LIN {X 0,Y 100.276,Z 426.301,A -85,B 0,C 180,E1 -26714.761,E2 -26714.761} C_VEL
LIN {X 0,Y 99.37,Z 433.159,A -85,B 0,C 180,E1 -26720.842,E2 -26720.842} C_VEL
LIN {X 0,Y 99.45,Z 437.817,A -85,B 0,C 180,E1 -26725.946,E2 -26725.946} C_VEL
LIN {X 0,Y 99.702,Z 440.8,A -85,B 0,C 180,E1 -26729.999,E2 -26729.999} C_VEL
LIN {X 0,Y 99.27,Z 443.094,A -85,B 0,C 180,E1 -26734.059,E2 -26734.059} C_VEL
LIN {X 0,Y 99.023,Z 444.925,A -85,B 0,C 180,E1 -26738.159,E2 -26738.159} C_VEL
LIN {X 0,Y 99.917,Z 447.345,A -85,B 0,C 180,E1 -26746.34,E2 -26746.34} C_VEL
LIN {X 0,Y 102.956,Z 448.359,A -85,B 0,C 180,E1 -26754.177,E2 -26754.177} C_VEL
LIN {X 0,Y 108.06,Z 448.023,A -85,B 0,C 180,E1 -26761.351,E2 -26761.351} C_VEL
LIN {X 0,Y 111.325,Z 447.297,A -85,B 0,C 180,E1 -26764.844,E2 -26764.844} C_VEL
LIN {X 0,Y 118.698,Z 444.902,A -85,B 0,C 180,E1 -26770.639,E2 -26770.639} C_VEL
LIN {X 0,Y 127.654,Z 441.015,A -85,B 0,C 180,E1 -26775.701,E2 -26775.701} C_VEL
LIN {X 0,Y 135.078,Z 437.071,A -85,B 0,C 180,E1 -26778.974,E2 -26778.974} C_VEL
LIN {X 0,Y 142.954,Z 432.141,A -85,B 0,C 180,E1 -26781.868,E2 -26781.868} C_VEL
LIN {X 0,Y 152.719,Z 424.964,A -85,B 0,C 180,E1 -26784.769,E2 -26784.769} C_VEL
LIN {X 0,Y 161.484,Z 417.418,A -85,B 0,C 180,E1 -26786.906,E2 -26786.906} C_VEL
LIN {X 0,Y 170.55,Z 408.157,A -85,B 0,C 180,E1 -26788.766,E2 -26788.766} C_VEL
LIN {X 0,Y 179.159,Z 397.683,A -85,B 0,C 180,E1 -26790.216,E2 -26790.216} C_VEL
LIN {X 0,Y 187.164,Z 385.927,A -85,B 0,C 180,E1 -26791.369,E2 -26791.369} C_VEL
LIN {X 0,Y 193.611,Z 374.263,A -85,B 0,C 180,E1 -26792.226,E2 -26792.226} C_VEL
LIN {X 0,Y 199.333,Z 361.205,A -85,B 0,C 180,E1 -26792.895,E2 -26792.895} C_VEL
LIN {X 0,Y 200.129,Z 359.001,A -85,B 0,C 180,E1 -26792.986,E2 -26792.986} C_VEL
LIN {X 0,Y 200.135,Z 358.847,A -85,B 0,C 180,E1 -26793.242,E2 -26793.242} C_VEL
LIN {X 0,Y 199.484,Z 360.339,A -85,B 0,C 180,E1 -26793.791,E2 -26793.791} C_VEL
LIN {X 0,Y 198.376,Z 362.917,A -85,B 0,C 180,E1 -26794.295,E2 -26794.295} C_VEL
LIN {X 0,Y 195.362,Z 369.602,A -85,B 0,C 180,E1 -26795.081,E2 -26795.081} C_VEL
LIN {X 0,Y 191.94,Z 376.275,A -85,B 0,C 180,E1 -26795.732,E2 -26795.732} C_VEL
LIN {X 0,Y 185.418,Z 386.983,A -85,B 0,C 180,E1 -26796.812,E2 -26796.812} C_VEL
LIN {X 0,Y 177.571,Z 397.49,A -85,B 0,C 180,E1 -26798.219,E2 -26798.219} C_VEL
LIN {X 0,Y 168.913,Z 406.976,A -85,B 0,C 180,E1 -26799.961,E2 -26799.961} C_VEL
LIN {X 0,Y 159.727,Z 415.31,A -85,B 0,C 180,E1 -26802.061,E2 -26802.061} C_VEL
LIN {X 0,Y 150.644,Z 422.152,A -85,B 0,C 180,E1 -26804.439,E2 -26804.439} C_VEL
LIN {X 0,Y 141.958,Z 427.534,A -85,B 0,C 180,E1 -26807.126,E2 -26807.126} C_VEL
LIN {X 0,Y 132.044,Z 432.427,A -85,B 0,C 180,E1 -26810.812,E2 -26810.812} C_VEL
LIN {X 0,Y 125.872,Z 434.856,A -85,B 0,C 180,E1 -26813.588,E2 -26813.588} C_VEL
LIN {X 0,Y 119.656,Z 436.729,A -85,B 0,C 180,E1 -26816.841,E2 -26816.841} C_VEL
LIN {X 0,Y 112.482,Z 438.152,A -85,B 0,C 180,E1 -26821.437,E2 -26821.437} C_VEL
LIN {X 0,Y 105.078,Z 438.534,A -85,B 0,C 180,E1 -26827.687,E2 -26827.687} C_VEL
LIN {X 0,Y 100.769,Z 437.945,A -85,B 0,C 180,E1 -26832.475,E2 -26832.475} C_VEL
LIN {X 0,Y 96.542,Z 436.3,A -85,B 0,C 180,E1 -26838.854,E2 -26838.854} C_VEL
LIN {X 0,Y 93.138,Z 433.039,A -85,B 0,C 180,E1 -26846.92,E2 -26846.92} C_VEL
LIN {X 0,Y 91.475,Z 428.303,A -85,B 0,C 180,E1 -26855.182,E2 -26855.182} C_VEL
LIN {X 0,Y 91.387,Z 423.638,A -85,B 0,C 180,E1 -26861.508,E2 -26861.508} C_VEL
LIN {X 0,Y 92.227,Z 417.856,A -85,B 0,C 180,E1 -26867.807,E2 -26867.807} C_VEL
LIN {X 0,Y 93.74,Z 410.783,A -85,B 0,C 180,E1 -26873.954,E2 -26873.954} C_VEL
LIN {X 0,Y 96.114,Z 401.66,A -85,B 0,C 180,E1 -26880.167,E2 -26880.167} C_VEL
LIN {X 0,Y 98.865,Z 392.134,A -85,B 0,C 180,E1 -26885.194,E2 -26885.194} C_VEL
LIN {X 0,Y 102.107,Z 380.518,A -85,B 0,C 180,E1 -26889.871,E2 -26889.871} C_VEL
LIN {X 0,Y 105.174,Z 368.48,A -85,B 0,C 180,E1 -26893.543,E2 -26893.543} C_VEL
LIN {X 0,Y 107.957,Z 355.625,A -85,B 0,C 180,E1 -26896.428,E2 -26896.428} C_VEL
LIN {X 0,Y 110.286,Z 342.25,A -85,B 0,C 180,E1 -26898.577,E2 -26898.577} C_VEL
LIN {X 0,Y 111.831,Z 328.48,A -85,B 0,C 180,E1 -26900.056,E2 -26900.056} C_VEL
LIN {X 0,Y 115.307,Z 288.804,A -85,B 0,C 180,E1 -26902.945,E2 -26902.945} C_VEL
LIN {X 0,Y 108.992,Z 272.53,A -85,B 0,C 180,E1 -26906.42,E2 -26906.42} C_VEL
LIN {X 0,Y 104.471,Z 262.113,A -85,B 0,C 180,E1 -26909.085,E2 -26909.085} C_VEL
LIN {X 0,Y 98.736,Z 250.528,A -85,B 0,C 180,E1 -26912.663,E2 -26912.663} C_VEL
LIN {X 0,Y 96.221,Z 246.747,A -85,B 0,C 180,E1 -26914.262,E2 -26914.262} C_VEL
LIN {X 0,Y 94.549,Z 244.182,A -85,B 0,C 180,E1 -26915.399,E2 -26915.399} C_VEL
LIN {X 0,Y 94.223,Z 242.747,A -85,B 0,C 180,E1 -26915.888,E2 -26915.888} C_VEL
LIN {X 0,Y 94.067,Z 242.767,A -85,B 0,C 180,E1 -26922.953,E2 -26922.953} C_VEL
LIN {X 0,Y 93.79,Z 242.798,A -85,B 0,C 180,E1 -26927.443,E2 -26927.443} C_VEL
LIN {X 0,Y 93.693,Z 242.786,A -85,B 0,C 180,E1 -26932.029,E2 -26932.029} C_VEL
LIN {X 0,Y 93.62,Z 242.82,A -85,B 0,C 180,E1 -26936.772,E2 -26936.772} C_VEL
LIN {X 0,Y 93.584,Z 242.8,A -85,B 0,C 180,E1 -26944.302,E2 -26944.302} C_VEL
LIN {X 0,Y 93.528,Z 242.815,A -85,B 0,C 180,E1 -26952.556,E2 -26952.556} C_VEL
LIN {X 0,Y 93.532,Z 242.834,A -85,B 0,C 180,E1 -26958.714,E2 -26958.714} C_VEL
LIN {X 0,Y 93.585,Z 242.821,A -85,B 0,C 180,E1 -26965.699,E2 -26965.699} C_VEL
LIN {X 0,Y 93.67,Z 242.801,A -85,B 0,C 180,E1 -26974.207,E2 -26974.207} C_VEL
LIN {X 0,Y 93.694,Z 242.81,A -85,B 0,C 180,E1 -26977.973,E2 -26977.973} C_VEL
LIN {X 0,Y 94.045,Z 242.733,A -85,B 0,C 180,E1 -26987.045,E2 -26987.045} C_VEL
LIN {X 0,Y 94.138,Z 242.707,A -85,B 0,C 180,E1 -26991.413,E2 -26991.413} C_VEL
LIN {X 0,Y 94.759,Z 242.681,A -85,B 0,C 180,E1 -27000,E2 -27000} C_VEL
LIN {X 0,Y 94.136,Z 242.725,A -85,B 0,C 180,E1 -27008.588,E2 -27008.588} C_VEL
LIN {X 0,Y 93.962,Z 242.78,A -85,B 0,C 180,E1 -27013.498,E2 -27013.498} C_VEL
LIN {X 0,Y 93.655,Z 242.802,A -85,B 0,C 180,E1 -27022.038,E2 -27022.038} C_VEL
LIN {X 0,Y 93.6,Z 242.83,A -85,B 0,C 180,E1 -27026.777,E2 -27026.777} C_VEL
LIN {X 0,Y 93.581,Z 242.953,A -85,B 0,C 180,E1 -27030.46,E2 -27030.46} C_VEL
LIN {X 0,Y 94.612,Z 245.714,A -85,B 0,C 180,E1 -27031.331,E2 -27031.331} C_VEL
LIN {X 0,Y 96.125,Z 247.852,A -85,B 0,C 180,E1 -27032.322,E2 -27032.322} C_VEL
LIN {X 0,Y 102.127,Z 258.497,A -85,B 0,C 180,E1 -27036.133,E2 -27036.133} C_VEL
LIN {X 0,Y 107.329,Z 272.747,A -85,B 0,C 180,E1 -27039.577,E2 -27039.577} C_VEL
LIN {X 0,Y 112.457,Z 289.346,A -85,B 0,C 180,E1 -27042.816,E2 -27042.816} C_VEL
LIN {X 0,Y 113.674,Z 316.74,A -85,B 0,C 180,E1 -27045.754,E2 -27045.754} C_VEL
LIN {X 0,Y 110.773,Z 348.84,A -85,B 0,C 180,E1 -27048.226,E2 -27048.226} C_VEL
LIN {X 0,Y 108.763,Z 363.104,A -85,B 0,C 180,E1 -27050.047,E2 -27050.047} C_VEL
LIN {X 0,Y 106.272,Z 375.199,A -85,B 0,C 180,E1 -27052.284,E2 -27052.284} C_VEL
LIN {X 0,Y 103.156,Z 387.718,A -85,B 0,C 180,E1 -27055.473,E2 -27055.473} C_VEL
LIN {X 0,Y 99.991,Z 399.014,A -85,B 0,C 180,E1 -27059.363,E2 -27059.363} C_VEL
LIN {X 0,Y 96.926,Z 409.601,A -85,B 0,C 180,E1 -27064.21,E2 -27064.21} C_VEL
LIN {X 0,Y 94.678,Z 418.278,A -85,B 0,C 180,E1 -27069.353,E2 -27069.353} C_VEL
LIN {X 0,Y 92.992,Z 426.684,A -85,B 0,C 180,E1 -27075.78,E2 -27075.78} C_VEL
LIN {X 0,Y 92.35,Z 434.065,A -85,B 0,C 180,E1 -27083.104,E2 -27083.104} C_VEL
LIN {X 0,Y 92.698,Z 439.38,A -85,B 0,C 180,E1 -27089.999,E2 -27089.999} C_VEL
LIN {X 0,Y 92.287,Z 441.774,A -85,B 0,C 180,E1 -27094.366,E2 -27094.366} C_VEL
LIN {X 0,Y 92.291,Z 445.203,A -85,B 0,C 180,E1 -27103.205,E2 -27103.205} C_VEL
LIN {X 0,Y 94.534,Z 447.195,A -85,B 0,C 180,E1 -27111.82,E2 -27111.82} C_VEL
LIN {X 0,Y 99.083,Z 447.77,A -85,B 0,C 180,E1 -27119.768,E2 -27119.768} C_VEL
LIN {X 0,Y 105.387,Z 446.981,A -85,B 0,C 180,E1 -27126.882,E2 -27126.882} C_VEL
LIN {X 0,Y 113.406,Z 444.856,A -85,B 0,C 180,E1 -27132.975,E2 -27132.975} C_VEL
LIN {X 0,Y 122.808,Z 441.311,A -85,B 0,C 180,E1 -27138.069,E2 -27138.069} C_VEL
LIN {X 0,Y 133.255,Z 436.16,A -85,B 0,C 180,E1 -27142.289,E2 -27142.289} C_VEL
LIN {X 0,Y 141.558,Z 431.209,A -85,B 0,C 180,E1 -27145.002,E2 -27145.002} C_VEL
LIN {X 0,Y 151.742,Z 424.029,A -85,B 0,C 180,E1 -27147.698,E2 -27147.698} C_VEL
LIN {X 0,Y 160.865,Z 416.375,A -85,B 0,C 180,E1 -27149.637,E2 -27149.637} C_VEL
LIN {X 0,Y 170.215,Z 407.055,A -85,B 0,C 180,E1 -27151.328,E2 -27151.328} C_VEL
LIN {X 0,Y 179.048,Z 396.59,A -85,B 0,C 180,E1 -27152.632,E2 -27152.632} C_VEL
LIN {X 0,Y 186.418,Z 386.056,A -85,B 0,C 180,E1 -27153.556,E2 -27153.556} C_VEL
LIN {X 0,Y 192.996,Z 374.507,A -85,B 0,C 180,E1 -27154.326,E2 -27154.326} C_VEL
LIN {X 0,Y 196.724,Z 366.706,A -85,B 0,C 180,E1 -27154.693,E2 -27154.693} C_VEL
LIN {X 0,Y 196.816,Z 366.436,A -85,B 0,C 180,E1 -27154.942,E2 -27154.942} C_VEL
LIN {X 0,Y 191.94,Z 376.275,A -85,B 0,C 180,E1 -27155.732,E2 -27155.732} C_VEL
LIN {X 0,Y 188.861,Z 381.616,A -85,B 0,C 180,E1 -27156.025,E2 -27156.025} C_VEL
LIN {X 0,Y 183.135,Z 390.296,A -85,B 0,C 180,E1 -27156.019,E2 -27156.019} C_VEL
LIN {X 0,Y 176.926,Z 398.26,A -85,B 0,C 180,E1 -27156.115,E2 -27156.115} C_VEL
LIN {X 0,Y 173.08,Z 402.614,A -85,B 0,C 180,E1 -27156.583,E2 -27156.583} C_VEL
LIN {X 0,Y 164.976,Z 410.619,A -85,B 0,C 180,E1 -27158.114,E2 -27158.114} C_VEL
LIN {X 0,Y 156.76,Z 417.411,A -85,B 0,C 180,E1 -27159.85,E2 -27159.85} C_VEL
LIN {X 0,Y 146.429,Z 424.498,A -85,B 0,C 180,E1 -27162.37,E2 -27162.37} C_VEL
LIN {X 0,Y 136.999,Z 429.751,A -85,B 0,C 180,E1 -27165.137,E2 -27165.137} C_VEL
LIN {X 0,Y 126.742,Z 434.216,A -85,B 0,C 180,E1 -27168.807,E2 -27168.807} C_VEL
LIN {X 0,Y 117.198,Z 437.169,A -85,B 0,C 180,E1 -27173.111,E2 -27173.111} C_VEL
LIN {X 0,Y 111.284,Z 438.41,A -85,B 0,C 180,E1 -27176.379,E2 -27176.379} C_VEL
LIN {X 0,Y 105.419,Z 439.093,A -85,B 0,C 180,E1 -27180.258,E2 -27180.258} C_VEL
LIN {X 0,Y 98.893,Z 439.04,A -85,B 0,C 180,E1 -27185.78,E2 -27185.78} C_VEL
LIN {X 0,Y 92.512,Z 437.673,A -85,B 0,C 180,E1 -27193.174,E2 -27193.174} C_VEL
LIN {X 0,Y 88.028,Z 435.022,A -85,B 0,C 180,E1 -27201.141,E2 -27201.141} C_VEL
LIN {X 0,Y 85.208,Z 430.979,A -85,B 0,C 180,E1 -27209.662,E2 -27209.662} C_VEL
LIN {X 0,Y 84.225,Z 425.417,A -85,B 0,C 180,E1 -27218.525,E2 -27218.525} C_VEL
LIN {X 0,Y 84.857,Z 418.976,A -85,B 0,C 180,E1 -27226.443,E2 -27226.443} C_VEL
LIN {X 0,Y 86.221,Z 412.464,A -85,B 0,C 180,E1 -27232.763,E2 -27232.763} C_VEL
LIN {X 0,Y 88.348,Z 404.204,A -85,B 0,C 180,E1 -27239.127,E2 -27239.127} C_VEL
LIN {X 0,Y 91.333,Z 394.023,A -85,B 0,C 180,E1 -27245.194,E2 -27245.194} C_VEL
LIN {X 0,Y 94.547,Z 383.203,A -85,B 0,C 180,E1 -27250.105,E2 -27250.105} C_VEL
LIN {X 0,Y 97.969,Z 370.789,A -85,B 0,C 180,E1 -27254.312,E2 -27254.312} C_VEL
LIN {X 0,Y 100.825,Z 358.533,A -85,B 0,C 180,E1 -27257.386,E2 -27257.386} C_VEL
LIN {X 0,Y 103.332,Z 345.504,A -85,B 0,C 180,E1 -27259.717,E2 -27259.717} C_VEL
LIN {X 0,Y 105.035,Z 332.632,A -85,B 0,C 180,E1 -27261.342,E2 -27261.342} C_VEL
LIN {X 0,Y 108.949,Z 290.428,A -85,B 0,C 180,E1 -27264.595,E2 -27264.595} C_VEL
LIN {X 0,Y 103.317,Z 275.707,A -85,B 0,C 180,E1 -27267.995,E2 -27267.995} C_VEL
LIN {X 0,Y 99.279,Z 266.162,A -85,B 0,C 180,E1 -27270.576,E2 -27270.576} C_VEL
LIN {X 0,Y 93.908,Z 255.049,A -85,B 0,C 180,E1 -27274.293,E2 -27274.293} C_VEL
LIN {X 0,Y 89.81,Z 248.588,A -85,B 0,C 180,E1 -27277.244,E2 -27277.244} C_VEL
LIN {X 0,Y 87.568,Z 245.397,A -85,B 0,C 180,E1 -27278.948,E2 -27278.948} C_VEL
LIN {X 0,Y 87.064,Z 243.638,A -85,B 0,C 180,E1 -27279.585,E2 -27279.585} C_VEL
LIN {X 0,Y 86.932,Z 243.656,A -85,B 0,C 180,E1 -27284.038,E2 -27284.038} C_VEL
LIN {X 0,Y 86.646,Z 243.676,A -85,B 0,C 180,E1 -27288.933,E2 -27288.933} C_VEL
LIN {X 0,Y 86.584,Z 243.696,A -85,B 0,C 180,E1 -27296.764,E2 -27296.764} C_VEL
LIN {X 0,Y 86.502,Z 243.667,A -85,B 0,C 180,E1 -27305.663,E2 -27305.663} C_VEL
LIN {X 0,Y 86.452,Z 243.698,A -85,B 0,C 180,E1 -27312.976,E2 -27312.976} C_VEL
LIN {X 0,Y 86.454,Z 243.713,A -85,B 0,C 180,E1 -27319.434,E2 -27319.434} C_VEL
LIN {X 0,Y 86.528,Z 243.698,A -85,B 0,C 180,E1 -27325.351,E2 -27325.351} C_VEL
LIN {X 0,Y 86.585,Z 243.686,A -85,B 0,C 180,E1 -27333.238,E2 -27333.238} C_VEL
LIN {X 0,Y 86.634,Z 243.691,A -85,B 0,C 180,E1 -27341.066,E2 -27341.066} C_VEL
LIN {X 0,Y 86.905,Z 243.631,A -85,B 0,C 180,E1 -27346.039,E2 -27346.039} C_VEL
LIN {X 0,Y 87.036,Z 243.588,A -85,B 0,C 180,E1 -27350.707,E2 -27350.707} C_VEL
LIN {X 0,Y 87.689,Z 243.562,A -85,B 0,C 180,E1 -27360,E2 -27360} C_VEL
LIN {X 0,Y 87.029,Z 243.612,A -85,B 0,C 180,E1 -27369.295,E2 -27369.295} C_VEL
LIN {X 0,Y 86.862,Z 243.666,A -85,B 0,C 180,E1 -27374.048,E2 -27374.048} C_VEL
LIN {X 0,Y 86.6,Z 243.686,A -85,B 0,C 180,E1 -27378.943,E2 -27378.943} C_VEL
LIN {X 0,Y 86.569,Z 243.706,A -85,B 0,C 180,E1 -27386.63,E2 -27386.63} C_VEL
LIN {X 0,Y 87.674,Z 246.767,A -85,B 0,C 180,E1 -27387.794,E2 -27387.794} C_VEL
LIN {X 0,Y 89.254,Z 248.872,A -85,B 0,C 180,E1 -27388.997,E2 -27388.997} C_VEL
LIN {X 0,Y 94.992,Z 258.752,A -85,B 0,C 180,E1 -27393.187,E2 -27393.187} C_VEL
LIN {X 0,Y 97.157,Z 263.103,A -85,B 0,C 180,E1 -27394.67,E2 -27394.67} C_VEL
LIN {X 0,Y 101.692,Z 275.807,A -85,B 0,C 180,E1 -27397.915,E2 -27397.915} C_VEL
LIN {X 0,Y 106.337,Z 291.462,A -85,B 0,C 180,E1 -27401.213,E2 -27401.213} C_VEL
LIN {X 0,Y 107.289,Z 317.248,A -85,B 0,C 180,E1 -27404.151,E2 -27404.151} C_VEL
LIN {X 0,Y 104.328,Z 348.396,A -85,B 0,C 180,E1 -27406.662,E2 -27406.662} C_VEL
LIN {X 0,Y 102.233,Z 362.635,A -85,B 0,C 180,E1 -27408.571,E2 -27408.571} C_VEL
LIN {X 0,Y 99.521,Z 375.221,A -85,B 0,C 180,E1 -27411.039,E2 -27411.039} C_VEL
LIN {X 0,Y 96.365,Z 387.295,A -85,B 0,C 180,E1 -27414.305,E2 -27414.305} C_VEL
LIN {X 0,Y 93.262,Z 397.922,A -85,B 0,C 180,E1 -27418.162,E2 -27418.162} C_VEL
LIN {X 0,Y 90.048,Z 408.6,A -85,B 0,C 180,E1 -27423.334,E2 -27423.334} C_VEL
LIN {X 0,Y 87.698,Z 417.351,A -85,B 0,C 180,E1 -27428.86,E2 -27428.86} C_VEL
LIN {X 0,Y 86.197,Z 424.565,A -85,B 0,C 180,E1 -27434.633,E2 -27434.633} C_VEL
LIN {X 0,Y 85.38,Z 430.937,A -85,B 0,C 180,E1 -27441.033,E2 -27441.033} C_VEL
LIN {X 0,Y 85.533,Z 436.217,A -85,B 0,C 180,E1 -27447.644,E2 -27447.644} C_VEL
LIN {X 0,Y 85.701,Z 437.789,A -85,B 0,C 180,E1 -27449.999,E2 -27449.999} C_VEL
LIN {X 0,Y 85.62,Z 439.178,A -85,B 0,C 180,E1 -27452.351,E2 -27452.351} C_VEL
LIN {X 0,Y 85.119,Z 442.431,A -85,B 0,C 180,E1 -27459.504,E2 -27459.504} C_VEL
LIN {X 0,Y 86.414,Z 445.336,A -85,B 0,C 180,E1 -27468.984,E2 -27468.984} C_VEL
LIN {X 0,Y 90.188,Z 446.848,A -85,B 0,C 180,E1 -27477.874,E2 -27477.874} C_VEL
LIN {X 0,Y 96.188,Z 447.042,A -85,B 0,C 180,E1 -27485.768,E2 -27485.768} C_VEL
LIN {X 0,Y 103.869,Z 445.862,A -85,B 0,C 180,E1 -27492.579,E2 -27492.579} C_VEL
LIN {X 0,Y 113.102,Z 443.318,A -85,B 0,C 180,E1 -27498.215,E2 -27498.215} C_VEL
LIN {X 0,Y 123.512,Z 439.354,A -85,B 0,C 180,E1 -27502.807,E2 -27502.807} C_VEL
LIN {X 0,Y 131.837,Z 435.344,A -85,B 0,C 180,E1 -27505.717,E2 -27505.717} C_VEL
LIN {X 0,Y 140.6,Z 430.338,A -85,B 0,C 180,E1 -27508.184,E2 -27508.184} C_VEL
LIN {X 0,Y 151.182,Z 423.12,A -85,B 0,C 180,E1 -27510.648,E2 -27510.648} C_VEL
LIN {X 0,Y 160.606,Z 415.471,A -85,B 0,C 180,E1 -27512.389,E2 -27512.389} C_VEL
LIN {X 0,Y 168.621,Z 407.822,A -85,B 0,C 180,E1 -27513.649,E2 -27513.649} C_VEL
LIN {X 0,Y 177.614,Z 397.607,A -85,B 0,C 180,E1 -27514.833,E2 -27514.833} C_VEL
LIN {X 0,Y 178.459,Z 396.55,A -85,B 0,C 180,E1 -27514.927,E2 -27514.927} C_VEL
LIN {X 0,Y 179.649,Z 394.979,A -85,B 0,C 180,E1 -27515.463,E2 -27515.463} C_VEL
LIN {X 0,Y 173.08,Z 402.614,A -85,B 0,C 180,E1 -27516.583,E2 -27516.583} C_VEL
LIN {X 0,Y 169.135,Z 406.745,A -85,B 0,C 180,E1 -27517.092,E2 -27517.092} C_VEL
LIN {X 0,Y 161.837,Z 413.399,A -85,B 0,C 180,E1 -27517.416,E2 -27517.416} C_VEL
LIN {X 0,Y 154.094,Z 419.458,A -85,B 0,C 180,E1 -27517.826,E2 -27517.826} C_VEL
LIN {X 0,Y 149.483,Z 422.584,A -85,B 0,C 180,E1 -27518.524,E2 -27518.524} C_VEL
LIN {X 0,Y 139.272,Z 428.505,A -85,B 0,C 180,E1 -27520.994,E2 -27520.994} C_VEL
LIN {X 0,Y 128.598,Z 433.377,A -85,B 0,C 180,E1 -27524.142,E2 -27524.142} C_VEL
LIN {X 0,Y 121.558,Z 435.872,A -85,B 0,C 180,E1 -27526.628,E2 -27526.628} C_VEL
LIN {X 0,Y 114.298,Z 437.858,A -85,B 0,C 180,E1 -27529.673,E2 -27529.673} C_VEL
LIN {X 0,Y 106.014,Z 439.331,A -85,B 0,C 180,E1 -27533.924,E2 -27533.924} C_VEL
LIN {X 0,Y 96.988,Z 439.798,A -85,B 0,C 180,E1 -27540,E2 -27540} C_VEL
LIN {X 0,Y 91.672,Z 439.326,A -85,B 0,C 180,E1 -27544.708,E2 -27544.708} C_VEL
LIN {X 0,Y 86.013,Z 437.823,A -85,B 0,C 180,E1 -27551.34,E2 -27551.34} C_VEL
LIN {X 0,Y 81.011,Z 434.663,A -85,B 0,C 180,E1 -27560.305,E2 -27560.305} C_VEL
LIN {X 0,Y 78.049,Z 430.194,A -85,B 0,C 180,E1 -27569.683,E2 -27569.683} C_VEL
LIN {X 0,Y 77.166,Z 424,A -85,B 0,C 180,E1 -27579.608,E2 -27579.608} C_VEL
LIN {X 0,Y 78.18,Z 416.558,A -85,B 0,C 180,E1 -27588.813,E2 -27588.813} C_VEL
LIN {X 0,Y 79.863,Z 409.168,A -85,B 0,C 180,E1 -27595.842,E2 -27595.842} C_VEL
LIN {X 0,Y 82.454,Z 400.112,A -85,B 0,C 180,E1 -27602.55,E2 -27602.55} C_VEL
LIN {X 0,Y 85.687,Z 389.92,A -85,B 0,C 180,E1 -27608.342,E2 -27608.342} C_VEL
LIN {X 0,Y 89.129,Z 378.496,A -85,B 0,C 180,E1 -27613.237,E2 -27613.237} C_VEL
LIN {X 0,Y 92.536,Z 366.042,A -85,B 0,C 180,E1 -27617.184,E2 -27617.184} C_VEL
LIN {X 0,Y 95.223,Z 354.416,A -85,B 0,C 180,E1 -27619.906,E2 -27619.906} C_VEL
LIN {X 0,Y 97.727,Z 340.442,A -85,B 0,C 180,E1 -27622.2,E2 -27622.2} C_VEL
LIN {X 0,Y 99.413,Z 326.296,A -85,B 0,C 180,E1 -27623.702,E2 -27623.702} C_VEL
LIN {X 0,Y 102.727,Z 292.201,A -85,B 0,C 180,E1 -27626.391,E2 -27626.391} C_VEL
LIN {X 0,Y 97.64,Z 278.779,A -85,B 0,C 180,E1 -27629.729,E2 -27629.729} C_VEL
LIN {X 0,Y 93.977,Z 269.807,A -85,B 0,C 180,E1 -27632.367,E2 -27632.367} C_VEL
LIN {X 0,Y 89.165,Z 259.563,A -85,B 0,C 180,E1 -27636.055,E2 -27636.055} C_VEL
LIN {X 0,Y 84.695,Z 252.673,A -85,B 0,C 180,E1 -27639.554,E2 -27639.554} C_VEL
LIN {X 0,Y 82.508,Z 249.126,A -85,B 0,C 180,E1 -27641.512,E2 -27641.512} C_VEL
LIN {X 0,Y 80.518,Z 246.662,A -85,B 0,C 180,E1 -27643.314,E2 -27643.314} C_VEL
LIN {X 0,Y 79.861,Z 244.536,A -85,B 0,C 180,E1 -27644.188,E2 -27644.188} C_VEL
LIN {X 0,Y 79.513,Z 244.552,A -85,B 0,C 180,E1 -27650.706,E2 -27650.706} C_VEL
LIN {X 0,Y 79.481,Z 244.584,A -85,B 0,C 180,E1 -27657.843,E2 -27657.843} C_VEL
LIN {X 0,Y 79.375,Z 244.586,A -85,B 0,C 180,E1 -27662.092,E2 -27662.092} C_VEL
LIN {X 0,Y 79.363,Z 244.547,A -85,B 0,C 180,E1 -27668.31,E2 -27668.31} C_VEL
LIN {X 0,Y 79.383,Z 244.591,A -85,B 0,C 180,E1 -27675.096,E2 -27675.096} C_VEL
LIN {X 0,Y 79.384,Z 244.58,A -85,B 0,C 180,E1 -27682.826,E2 -27682.826} C_VEL
LIN {X 0,Y 79.376,Z 244.597,A -85,B 0,C 180,E1 -27687.911,E2 -27687.911} C_VEL
LIN {X 0,Y 79.526,Z 244.562,A -85,B 0,C 180,E1 -27693.777,E2 -27693.777} C_VEL
LIN {X 0,Y 79.507,Z 244.58,A -85,B 0,C 180,E1 -27699.294,E2 -27699.294} C_VEL
LIN {X 0,Y 79.81,Z 244.516,A -85,B 0,C 180,E1 -27705.622,E2 -27705.622} C_VEL
LIN {X 0,Y 79.927,Z 244.472,A -85,B 0,C 180,E1 -27709.872,E2 -27709.872} C_VEL
LIN {X 0,Y 80.618,Z 244.443,A -85,B 0,C 180,E1 -27720,E2 -27720} C_VEL
LIN {X 0,Y 79.914,Z 244.501,A -85,B 0,C 180,E1 -27730.131,E2 -27730.131} C_VEL
LIN {X 0,Y 79.689,Z 244.562,A -85,B 0,C 180,E1 -27735.342,E2 -27735.342} C_VEL
LIN {X 0,Y 79.478,Z 244.603,A -85,B 0,C 180,E1 -27742.075,E2 -27742.075} C_VEL
LIN {X 0,Y 80.354,Z 247.214,A -85,B 0,C 180,E1 -27743.178,E2 -27743.178} C_VEL
LIN {X 0,Y 82.439,Z 249.882,A -85,B 0,C 180,E1 -27745.062,E2 -27745.062} C_VEL
LIN {X 0,Y 88.612,Z 260.241,A -85,B 0,C 180,E1 -27750.249,E2 -27750.249} C_VEL
LIN {X 0,Y 92.09,Z 267.154,A -85,B 0,C 180,E1 -27752.932,E2 -27752.932} C_VEL
LIN {X 0,Y 96.736,Z 280.936,A -85,B 0,C 180,E1 -27756.649,E2 -27756.649} C_VEL
LIN {X 0,Y 100.267,Z 293.315,A -85,B 0,C 180,E1 -27759.376,E2 -27759.376} C_VEL
LIN {X 0,Y 100.964,Z 317.979,A -85,B 0,C 180,E1 -27762.361,E2 -27762.361} C_VEL
LIN {X 0,Y 97.966,Z 347.941,A -85,B 0,C 180,E1 -27764.891,E2 -27764.891} C_VEL
LIN {X 0,Y 95.78,Z 362.167,A -85,B 0,C 180,E1 -27766.895,E2 -27766.895} C_VEL
LIN {X 0,Y 92.884,Z 375.031,A -85,B 0,C 180,E1 -27769.563,E2 -27769.563} C_VEL
LIN {X 0,Y 89.435,Z 387.51,A -85,B 0,C 180,E1 -27773.187,E2 -27773.187} C_VEL
LIN {X 0,Y 85.849,Z 399.05,A -85,B 0,C 180,E1 -27777.85,E2 -27777.85} C_VEL
LIN {X 0,Y 82.63,Z 409.408,A -85,B 0,C 180,E1 -27783.477,E2 -27783.477} C_VEL
LIN {X 0,Y 80.361,Z 417.886,A -85,B 0,C 180,E1 -27789.522,E2 -27789.522} C_VEL
LIN {X 0,Y 78.75,Z 426.083,A -85,B 0,C 180,E1 -27797.107,E2 -27797.107} C_VEL
LIN {X 0,Y 78.419,Z 432.634,A -85,B 0,C 180,E1 -27804.857,E2 -27804.857} C_VEL
LIN {X 0,Y 78.701,Z 436.18,A -85,B 0,C 180,E1 -27809.999,E2 -27809.999} C_VEL
LIN {X 0,Y 78.697,Z 437.639,A -85,B 0,C 180,E1 -27812.558,E2 -27812.558} C_VEL
LIN {X 0,Y 78.234,Z 441.069,A -85,B 0,C 180,E1 -27820.349,E2 -27820.349} C_VEL
LIN {X 0,Y 79.763,Z 444.243,A -85,B 0,C 180,E1 -27830.635,E2 -27830.635} C_VEL
LIN {X 0,Y 83.981,Z 446.021,A -85,B 0,C 180,E1 -27840.139,E2 -27840.139} C_VEL
LIN {X 0,Y 90.507,Z 446.445,A -85,B 0,C 180,E1 -27848.403,E2 -27848.403} C_VEL
LIN {X 0,Y 94.396,Z 446.162,A -85,B 0,C 180,E1 -27852.071,E2 -27852.071} C_VEL
LIN {X 0,Y 103.461,Z 444.619,A -85,B 0,C 180,E1 -27858.349,E2 -27858.349} C_VEL
LIN {X 0,Y 113.833,Z 441.723,A -85,B 0,C 180,E1 -27863.379,E2 -27863.379} C_VEL
LIN {X 0,Y 125.11,Z 437.315,A -85,B 0,C 180,E1 -27867.416,E2 -27867.416} C_VEL
LIN {X 0,Y 133.98,Z 432.968,A -85,B 0,C 180,E1 -27869.94,E2 -27869.94} C_VEL
LIN {X 0,Y 144.74,Z 426.631,A -85,B 0,C 180,E1 -27872.391,E2 -27872.391} C_VEL
LIN {X 0,Y 154.271,Z 419.878,A -85,B 0,C 180,E1 -27874.122,E2 -27874.122} C_VEL
LIN {X 0,Y 162.359,Z 413.137,A -85,B 0,C 180,E1 -27875.37,E2 -27875.37} C_VEL
LIN {X 0,Y 161.415,Z 413.848,A -85,B 0,C 180,E1 -27876.11,E2 -27876.11} C_VEL
LIN {X 0,Y 151.16,Z 421.501,A -85,B 0,C 180,E1 -27878.164,E2 -27878.164} C_VEL
LIN {X 0,Y 149.483,Z 422.584,A -85,B 0,C 180,E1 -27878.524,E2 -27878.524} C_VEL
LIN {X 0,Y 144.737,Z 425.531,A -85,B 0,C 180,E1 -27879.309,E2 -27879.309} C_VEL
LIN {X 0,Y 136.15,Z 430.119,A -85,B 0,C 180,E1 -27880.11,E2 -27880.11} C_VEL
LIN {X 0,Y 127.366,Z 433.963,A -85,B 0,C 180,E1 -27881.11,E2 -27881.11} C_VEL
LIN {X 0,Y 122.374,Z 435.711,A -85,B 0,C 180,E1 -27882.277,E2 -27882.277} C_VEL
LIN {X 0,Y 113.038,Z 438.307,A -85,B 0,C 180,E1 -27885.599,E2 -27885.599} C_VEL
LIN {X 0,Y 106.221,Z 439.577,A -85,B 0,C 180,E1 -27888.551,E2 -27888.551} C_VEL
LIN {X 0,Y 99.325,Z 440.327,A -85,B 0,C 180,E1 -27892.133,E2 -27892.133} C_VEL
LIN {X 0,Y 91.462,Z 440.36,A -85,B 0,C 180,E1 -27897.321,E2 -27897.321} C_VEL
LIN {X 0,Y 83.169,Z 439.061,A -85,B 0,C 180,E1 -27904.847,E2 -27904.847} C_VEL
LIN {X 0,Y 77.009,Z 436.551,A -85,B 0,C 180,E1 -27913.192,E2 -27913.192} C_VEL
LIN {X 0,Y 72.66,Z 432.709,A -85,B 0,C 180,E1 -27922.761,E2 -27922.761} C_VEL
LIN {X 0,Y 70.896,Z 429.246,A -85,B 0,C 180,E1 -27929.712,E2 -27929.712} C_VEL
LIN {X 0,Y 70.111,Z 423.837,A -85,B 0,C 180,E1 -27938.792,E2 -27938.792} C_VEL
LIN {X 0,Y 71.022,Z 416.549,A -85,B 0,C 180,E1 -27948.508,E2 -27948.508} C_VEL
LIN {X 0,Y 72.836,Z 408.74,A -85,B 0,C 180,E1 -27956.536,E2 -27956.536} C_VEL
LIN {X 0,Y 75.653,Z 399.383,A -85,B 0,C 180,E1 -27963.964,E2 -27963.964} C_VEL
LIN {X 0,Y 79.064,Z 389.182,A -85,B 0,C 180,E1 -27970.061,E2 -27970.061} C_VEL
LIN {X 0,Y 82.782,Z 377.425,A -85,B 0,C 180,E1 -27975.246,E2 -27975.246} C_VEL
LIN {X 0,Y 86.252,Z 365.208,A -85,B 0,C 180,E1 -27979.219,E2 -27979.219} C_VEL
LIN {X 0,Y 89.4,Z 351.682,A -85,B 0,C 180,E1 -27982.338,E2 -27982.338} C_VEL
LIN {X 0,Y 91.715,Z 338.672,A -85,B 0,C 180,E1 -27984.421,E2 -27984.421} C_VEL
LIN {X 0,Y 93.666,Z 321.422,A -85,B 0,C 180,E1 -27986.127,E2 -27986.127} C_VEL
LIN {X 0,Y 96.39,Z 293.602,A -85,B 0,C 180,E1 -27988.449,E2 -27988.449} C_VEL
LIN {X 0,Y 91.431,Z 280.084,A -85,B 0,C 180,E1 -27992.192,E2 -27992.192} C_VEL
LIN {X 0,Y 87.336,Z 270.29,A -85,B 0,C 180,E1 -27995.492,E2 -27995.492} C_VEL
LIN {X 0,Y 84.491,Z 264.089,A -85,B 0,C 180,E1 -27997.938,E2 -27997.938} C_VEL
LIN {X 0,Y 78.699,Z 254.69,A -85,B 0,C 180,E1 -28003.255,E2 -28003.255} C_VEL
LIN {X 0,Y 76.383,Z 251.503,A -85,B 0,C 180,E1 -28005.607,E2 -28005.607} C_VEL
LIN {X 0,Y 75.775,Z 250.503,A -85,B 0,C 180,E1 -28006.289,E2 -28006.289} C_VEL
LIN {X 0,Y 73.453,Z 248.246,A -85,B 0,C 180,E1 -28008.748,E2 -28008.748} C_VEL
LIN {X 0,Y 72.475,Z 245.429,A -85,B 0,C 180,E1 -28010.399,E2 -28010.399} C_VEL
LIN {X 0,Y 72.358,Z 245.473,A -85,B 0,C 180,E1 -28019.056,E2 -28019.056} C_VEL
LIN {X 0,Y 72.292,Z 245.433,A -85,B 0,C 180,E1 -28025.685,E2 -28025.685} C_VEL
LIN {X 0,Y 72.243,Z 245.465,A -85,B 0,C 180,E1 -28032.922,E2 -28032.922} C_VEL
LIN {X 0,Y 72.292,Z 245.469,A -85,B 0,C 180,E1 -28041.056,E2 -28041.056} C_VEL
LIN {X 0,Y 72.293,Z 245.465,A -85,B 0,C 180,E1 -28044.318,E2 -28044.318} C_VEL
LIN {X 0,Y 72.359,Z 245.467,A -85,B 0,C 180,E1 -28050.946,E2 -28050.946} C_VEL
LIN {X 0,Y 72.391,Z 245.459,A -85,B 0,C 180,E1 -28057.149,E2 -28057.149} C_VEL
LIN {X 0,Y 72.71,Z 245.402,A -85,B 0,C 180,E1 -28065.153,E2 -28065.153} C_VEL
LIN {X 0,Y 72.828,Z 245.357,A -85,B 0,C 180,E1 -28068.872,E2 -28068.872} C_VEL
LIN {X 0,Y 73.546,Z 245.324,A -85,B 0,C 180,E1 -28080,E2 -28080} C_VEL
LIN {X 0,Y 72.81,Z 245.392,A -85,B 0,C 180,E1 -28091.131,E2 -28091.131} C_VEL
LIN {X 0,Y 72.58,Z 245.65,A -85,B 0,C 180,E1 -28096.367,E2 -28096.367} C_VEL
LIN {X 0,Y 73.505,Z 248.315,A -85,B 0,C 180,E1 -28097.799,E2 -28097.799} C_VEL
LIN {X 0,Y 75.71,Z 250.936,A -85,B 0,C 180,E1 -28100.23,E2 -28100.23} C_VEL
LIN {X 0,Y 77.849,Z 254.304,A -85,B 0,C 180,E1 -28102.562,E2 -28102.562} C_VEL
LIN {X 0,Y 83.309,Z 263.656,A -85,B 0,C 180,E1 -28107.773,E2 -28107.773} C_VEL
LIN {X 0,Y 87.075,Z 271.144,A -85,B 0,C 180,E1 -28110.967,E2 -28110.967} C_VEL
LIN {X 0,Y 91.459,Z 284.893,A -85,B 0,C 180,E1 -28114.951,E2 -28114.951} C_VEL
LIN {X 0,Y 94.259,Z 295.203,A -85,B 0,C 180,E1 -28117.407,E2 -28117.407} C_VEL
LIN {X 0,Y 94.779,Z 318.003,A -85,B 0,C 180,E1 -28120.334,E2 -28120.334} C_VEL
LIN {X 0,Y 91.61,Z 347.954,A -85,B 0,C 180,E1 -28123.011,E2 -28123.011} C_VEL
LIN {X 0,Y 89.454,Z 361.304,A -85,B 0,C 180,E1 -28124.999,E2 -28124.999} C_VEL
LIN {X 0,Y 86.297,Z 374.647,A -85,B 0,C 180,E1 -28127.912,E2 -28127.912} C_VEL
LIN {X 0,Y 82.564,Z 387.447,A -85,B 0,C 180,E1 -28131.891,E2 -28131.891} C_VEL
LIN {X 0,Y 78.84,Z 398.889,A -85,B 0,C 180,E1 -28136.905,E2 -28136.905} C_VEL
LIN {X 0,Y 75.807,Z 408.223,A -85,B 0,C 180,E1 -28142.382,E2 -28142.382} C_VEL
LIN {X 0,Y 73.388,Z 416.817,A -85,B 0,C 180,E1 -28148.952,E2 -28148.952} C_VEL
LIN {X 0,Y 71.917,Z 423.887,A -85,B 0,C 180,E1 -28155.857,E2 -28155.857} C_VEL
LIN {X 0,Y 71.416,Z 430.75,A -85,B 0,C 180,E1 -28164.351,E2 -28164.351} C_VEL
LIN {X 0,Y 71.711,Z 434.451,A -85,B 0,C 180,E1 -28169.998,E2 -28169.998} C_VEL
LIN {X 0,Y 71.796,Z 436.022,A -85,B 0,C 180,E1 -28172.804,E2 -28172.804} C_VEL
LIN {X 0,Y 71.375,Z 439.65,A -85,B 0,C 180,E1 -28181.356,E2 -28181.356} C_VEL
LIN {X 0,Y 73.232,Z 443.069,A -85,B 0,C 180,E1 -28192.572,E2 -28192.572} C_VEL
LIN {X 0,Y 77.938,Z 445.098,A -85,B 0,C 180,E1 -28202.753,E2 -28202.753} C_VEL
LIN {X 0,Y 85.043,Z 445.828,A -85,B 0,C 180,E1 -28211.384,E2 -28211.384} C_VEL
LIN {X 0,Y 93.891,Z 445.218,A -85,B 0,C 180,E1 -28218.461,E2 -28218.461} C_VEL
LIN {X 0,Y 104.196,Z 443.298,A -85,B 0,C 180,E1 -28224.036,E2 -28224.036} C_VEL
LIN {X 0,Y 115.496,Z 440.003,A -85,B 0,C 180,E1 -28228.418,E2 -28228.418} C_VEL
LIN {X 0,Y 127.49,Z 435.252,A -85,B 0,C 180,E1 -28231.884,E2 -28231.884} C_VEL
LIN {X 0,Y 136.87,Z 430.581,A -85,B 0,C 180,E1 -28233.972,E2 -28233.972} C_VEL
LIN {X 0,Y 146.458,Z 424.831,A -85,B 0,C 180,E1 -28235.745,E2 -28235.745} C_VEL
LIN {X 0,Y 145.834,Z 425.128,A -85,B 0,C 180,E1 -28236.295,E2 -28236.295} C_VEL
LIN {X 0,Y 135.236,Z 430.667,A -85,B 0,C 180,E1 -28238.667,E2 -28238.667} C_VEL
LIN {X 0,Y 123.58,Z 435.335,A -85,B 0,C 180,E1 -28241.898,E2 -28241.898} C_VEL
LIN {X 0,Y 122.374,Z 435.711,A -85,B 0,C 180,E1 -28242.277,E2 -28242.277} C_VEL
LIN {X 0,Y 117.331,Z 437.251,A -85,B 0,C 180,E1 -28243.582,E2 -28243.582} C_VEL
LIN {X 0,Y 108.204,Z 439.423,A -85,B 0,C 180,E1 -28245.244,E2 -28245.244} C_VEL
LIN {X 0,Y 99.129,Z 440.754,A -85,B 0,C 180,E1 -28247.263,E2 -28247.263} C_VEL
LIN {X 0,Y 94.279,Z 441.047,A -85,B 0,C 180,E1 -28249.226,E2 -28249.226} C_VEL
LIN {X 0,Y 84.599,Z 440.672,A -85,B 0,C 180,E1 -28255.469,E2 -28255.469} C_VEL
LIN {X 0,Y 77.351,Z 439.267,A -85,B 0,C 180,E1 -28261.948,E2 -28261.948} C_VEL
LIN {X 0,Y 70.185,Z 436.163,A -85,B 0,C 180,E1 -28271.552,E2 -28271.552} C_VEL
LIN {X 0,Y 65.56,Z 431.873,A -85,B 0,C 180,E1 -28282.033,E2 -28282.033} C_VEL
LIN {X 0,Y 63.586,Z 427.558,A -85,B 0,C 180,E1 -28290.858,E2 -28290.858} C_VEL
LIN {X 0,Y 63.151,Z 421.033,A -85,B 0,C 180,E1 -28301.892,E2 -28301.892} C_VEL
LIN {X 0,Y 64.555,Z 413.346,A -85,B 0,C 180,E1 -28311.975,E2 -28311.975} C_VEL
LIN {X 0,Y 67.112,Z 404.088,A -85,B 0,C 180,E1 -28321.188,E2 -28321.188} C_VEL
LIN {X 0,Y 70.626,Z 393.671,A -85,B 0,C 180,E1 -28328.891,E2 -28328.891} C_VEL
LIN {X 0,Y 74.526,Z 382.373,A -85,B 0,C 180,E1 -28334.971,E2 -28334.971} C_VEL
LIN {X 0,Y 78.313,Z 370.443,A -85,B 0,C 180,E1 -28339.662,E2 -28339.662} C_VEL
LIN {X 0,Y 81.686,Z 357.871,A -85,B 0,C 180,E1 -28343.207,E2 -28343.207} C_VEL
LIN {X 0,Y 84.563,Z 344.717,A -85,B 0,C 180,E1 -28345.797,E2 -28345.797} C_VEL
LIN {X 0,Y 86.541,Z 330.722,A -85,B 0,C 180,E1 -28347.622,E2 -28347.622} C_VEL
LIN {X 0,Y 90.328,Z 295.351,A -85,B 0,C 180,E1 -28350.691,E2 -28350.691} C_VEL
LIN {X 0,Y 84.512,Z 279.253,A -85,B 0,C 180,E1 -28355.676,E2 -28355.676} C_VEL
LIN {X 0,Y 79.803,Z 268.429,A -85,B 0,C 180,E1 -28360.146,E2 -28360.146} C_VEL
LIN {X 0,Y 74.429,Z 259.627,A -85,B 0,C 180,E1 -28365.661,E2 -28365.661} C_VEL
LIN {X 0,Y 71.936,Z 256.072,A -85,B 0,C 180,E1 -28368.535,E2 -28368.535} C_VEL
LIN {X 0,Y 69.58,Z 253.067,A -85,B 0,C 180,E1 -28371.542,E2 -28371.542} C_VEL
LIN {X 0,Y 68.672,Z 251.49,A -85,B 0,C 180,E1 -28372.916,E2 -28372.916} C_VEL
LIN {X 0,Y 66.313,Z 249.32,A -85,B 0,C 180,E1 -28376.337,E2 -28376.337} C_VEL
LIN {X 0,Y 65.363,Z 246.879,A -85,B 0,C 180,E1 -28378.284,E2 -28378.284} C_VEL
LIN {X 0,Y 65.301,Z 246.352,A -85,B 0,C 180,E1 -28378.752,E2 -28378.752} C_VEL
LIN {X 0,Y 65.199,Z 246.315,A -85,B 0,C 180,E1 -28390.3,E2 -28390.3} C_VEL
LIN {X 0,Y 65.2,Z 246.359,A -85,B 0,C 180,E1 -28399.703,E2 -28399.703} C_VEL
LIN {X 0,Y 65.242,Z 246.357,A -85,B 0,C 180,E1 -28409.519,E2 -28409.519} C_VEL
LIN {X 0,Y 65.228,Z 246.342,A -85,B 0,C 180,E1 -28414.471,E2 -28414.471} C_VEL
LIN {X 0,Y 65.609,Z 246.289,A -85,B 0,C 180,E1 -28424.603,E2 -28424.603} C_VEL
LIN {X 0,Y 65.733,Z 246.245,A -85,B 0,C 180,E1 -28427.653,E2 -28427.653} C_VEL
LIN {X 0,Y 66.443,Z 246.209,A -85,B 0,C 180,E1 -28440,E2 -28440} C_VEL
LIN {X 0,Y 65.773,Z 246.309,A -85,B 0,C 180,E1 -28448.643,E2 -28448.643} C_VEL
LIN {X 0,Y 66.615,Z 248.881,A -85,B 0,C 180,E1 -28450.448,E2 -28450.448} C_VEL
LIN {X 0,Y 68.72,Z 251.302,A -85,B 0,C 180,E1 -28453.594,E2 -28453.594} C_VEL
LIN {X 0,Y 71.042,Z 255.262,A -85,B 0,C 180,E1 -28456.898,E2 -28456.898} C_VEL
LIN {X 0,Y 72.32,Z 257.092,A -85,B 0,C 180,E1 -28458.493,E2 -28458.493} C_VEL
LIN {X 0,Y 76.104,Z 263.236,A -85,B 0,C 180,E1 -28462.837,E2 -28462.837} C_VEL
LIN {X 0,Y 80.971,Z 272.512,A -85,B 0,C 180,E1 -28467.743,E2 -28467.743} C_VEL
LIN {X 0,Y 82.898,Z 277.592,A -85,B 0,C 180,E1 -28469.649,E2 -28469.649} C_VEL
LIN {X 0,Y 86.949,Z 291.528,A -85,B 0,C 180,E1 -28473.759,E2 -28473.759} C_VEL
LIN {X 0,Y 88.35,Z 297.455,A -85,B 0,C 180,E1 -28475.221,E2 -28475.221} C_VEL
LIN {X 0,Y 88.674,Z 318,A -85,B 0,C 180,E1 -28478.062,E2 -28478.062} C_VEL
LIN {X 0,Y 85.355,Z 347.74,A -85,B 0,C 180,E1 -28480.848,E2 -28480.848} C_VEL
LIN {X 0,Y 82.921,Z 361.784,A -85,B 0,C 180,E1 -28483.081,E2 -28483.081} C_VEL
LIN {X 0,Y 79.738,Z 374.432,A -85,B 0,C 180,E1 -28486.043,E2 -28486.043} C_VEL
LIN {X 0,Y 76.22,Z 385.922,A -85,B 0,C 180,E1 -28489.799,E2 -28489.799} C_VEL
LIN {X 0,Y 72.668,Z 396.445,A -85,B 0,C 180,E1 -28494.528,E2 -28494.528} C_VEL
LIN {X 0,Y 69.008,Z 407.035,A -85,B 0,C 180,E1 -28501.067,E2 -28501.067} C_VEL
LIN {X 0,Y 66.442,Z 415.69,A -85,B 0,C 180,E1 -28508.269,E2 -28508.269} C_VEL
LIN {X 0,Y 64.912,Z 422.813,A -85,B 0,C 180,E1 -28515.899,E2 -28515.899} C_VEL
LIN {X 0,Y 64.479,Z 429.759,A -85,B 0,C 180,E1 -28525.309,E2 -28525.309} C_VEL
LIN {X 0,Y 64.885,Z 434.288,A -85,B 0,C 180,E1 -28533.103,E2 -28533.103} C_VEL
LIN {X 0,Y 64.573,Z 438.13,A -85,B 0,C 180,E1 -28542.571,E2 -28542.571} C_VEL
LIN {X 0,Y 66.795,Z 441.841,A -85,B 0,C 180,E1 -28554.888,E2 -28554.888} C_VEL
LIN {X 0,Y 72.091,Z 444.128,A -85,B 0,C 180,E1 -28565.796,E2 -28565.796} C_VEL
LIN {X 0,Y 79.842,Z 445.103,A -85,B 0,C 180,E1 -28574.762,E2 -28574.762} C_VEL
LIN {X 0,Y 89.332,Z 444.795,A -85,B 0,C 180,E1 -28581.879,E2 -28581.879} C_VEL
LIN {X 0,Y 100.187,Z 443.209,A -85,B 0,C 180,E1 -28587.327,E2 -28587.327} C_VEL
LIN {X 0,Y 111.951,Z 440.27,A -85,B 0,C 180,E1 -28591.507,E2 -28591.507} C_VEL
LIN {X 0,Y 124.317,Z 435.86,A -85,B 0,C 180,E1 -28594.758,E2 -28594.758} C_VEL
LIN {X 0,Y 130.697,Z 433.062,A -85,B 0,C 180,E1 -28596.083,E2 -28596.083} C_VEL
LIN {X 0,Y 130.316,Z 433.171,A -85,B 0,C 180,E1 -28596.463,E2 -28596.463} C_VEL
LIN {X 0,Y 118.873,Z 437.088,A -85,B 0,C 180,E1 -28599.423,E2 -28599.423} C_VEL
LIN {X 0,Y 110.858,Z 439.084,A -85,B 0,C 180,E1 -28601.976,E2 -28601.976} C_VEL
LIN {X 0,Y 101.554,Z 440.563,A -85,B 0,C 180,E1 -28605.661,E2 -28605.661} C_VEL
LIN {X 0,Y 94.279,Z 441.047,A -85,B 0,C 180,E1 -28609.226,E2 -28609.226} C_VEL
LIN {X 0,Y 89.524,Z 441.118,A -85,B 0,C 180,E1 -28611.416,E2 -28611.416} C_VEL
LIN {X 0,Y 80.85,Z 440.675,A -85,B 0,C 180,E1 -28614.645,E2 -28614.645} C_VEL
LIN {X 0,Y 72.574,Z 439.443,A -85,B 0,C 180,E1 -28618.614,E2 -28618.614} C_VEL
LIN {X 0,Y 68.627,Z 438.259,A -85,B 0,C 180,E1 -28622.054,E2 -28622.054} C_VEL
LIN {X 0,Y 61.555,Z 434.258,A -85,B 0,C 180,E1 -28633.199,E2 -28633.199} C_VEL
LIN {X 0,Y 57.4,Z 429.024,A -85,B 0,C 180,E1 -28645.336,E2 -28645.336} C_VEL
LIN {X 0,Y 56.008,Z 422.005,A -85,B 0,C 180,E1 -28658.859,E2 -28658.859} C_VEL
LIN {X 0,Y 57.053,Z 414.625,A -85,B 0,C 180,E1 -28670.168,E2 -28670.168} C_VEL
LIN {X 0,Y 59.225,Z 406.494,A -85,B 0,C 180,E1 -28679.706,E2 -28679.706} C_VEL
LIN {X 0,Y 62.088,Z 398.09,A -85,B 0,C 180,E1 -28687.224,E2 -28687.224} C_VEL
LIN {X 0,Y 65.811,Z 388.034,A -85,B 0,C 180,E1 -28693.967,E2 -28693.967} C_VEL
LIN {X 0,Y 69.407,Z 377.835,A -85,B 0,C 180,E1 -28699.058,E2 -28699.058} C_VEL
LIN {X 0,Y 73.052,Z 366.492,A -85,B 0,C 180,E1 -28703.233,E2 -28703.233} C_VEL
LIN {X 0,Y 76.501,Z 353.5,A -85,B 0,C 180,E1 -28706.614,E2 -28706.614} C_VEL
LIN {X 0,Y 79.178,Z 340.402,A -85,B 0,C 180,E1 -28708.965,E2 -28708.965} C_VEL
LIN {X 0,Y 81.309,Z 324.161,A -85,B 0,C 180,E1 -28710.767,E2 -28710.767} C_VEL
LIN {X 0,Y 84.32,Z 296.815,A -85,B 0,C 180,E1 -28713.246,E2 -28713.246} C_VEL
LIN {X 0,Y 79.202,Z 282.285,A -85,B 0,C 180,E1 -28718.262,E2 -28718.262} C_VEL
LIN {X 0,Y 74.981,Z 272.208,A -85,B 0,C 180,E1 -28722.907,E2 -28722.907} C_VEL
LIN {X 0,Y 70.361,Z 264.566,A -85,B 0,C 180,E1 -28728.226,E2 -28728.226} C_VEL
LIN {X 0,Y 68.437,Z 261.697,A -85,B 0,C 180,E1 -28730.779,E2 -28730.779} C_VEL
LIN {X 0,Y 66.07,Z 258.277,A -85,B 0,C 180,E1 -28734.322,E2 -28734.322} C_VEL
LIN {X 0,Y 65.072,Z 257.156,A -85,B 0,C 180,E1 -28735.878,E2 -28735.878} C_VEL
LIN {X 0,Y 62.847,Z 254.237,A -85,B 0,C 180,E1 -28739.804,E2 -28739.804} C_VEL
LIN {X 0,Y 62.177,Z 252.766,A -85,B 0,C 180,E1 -28741.319,E2 -28741.319} C_VEL
LIN {X 0,Y 59.518,Z 250.783,A -85,B 0,C 180,E1 -28747.056,E2 -28747.056} C_VEL
LIN {X 0,Y 58.141,Z 247.682,A -85,B 0,C 180,E1 -28751.861,E2 -28751.861} C_VEL
LIN {X 0,Y 58.022,Z 247.226,A -85,B 0,C 180,E1 -28752.729,E2 -28752.729} C_VEL
LIN {X 0,Y 58.022,Z 247.24,A -85,B 0,C 180,E1 -28762.726,E2 -28762.726} C_VEL
LIN {X 0,Y 58.14,Z 247.236,A -85,B 0,C 180,E1 -28771.085,E2 -28771.085} C_VEL
LIN {X 0,Y 58.504,Z 247.176,A -85,B 0,C 180,E1 -28783.959,E2 -28783.959} C_VEL
LIN {X 0,Y 58.777,Z 247.11,A -85,B 0,C 180,E1 -28793.133,E2 -28793.133} C_VEL
LIN {X 0,Y 59.022,Z 247.282,A -85,B 0,C 180,E1 -28796.801,E2 -28796.801} C_VEL
LIN {X 0,Y 61.162,Z 251.362,A -85,B 0,C 180,E1 -28802.882,E2 -28802.882} C_VEL
LIN {X 0,Y 62.841,Z 252.914,A -85,B 0,C 180,E1 -28806.22,E2 -28806.22} C_VEL
LIN {X 0,Y 64.952,Z 256.583,A -85,B 0,C 180,E1 -28810.322,E2 -28810.322} C_VEL
LIN {X 0,Y 65.904,Z 257.994,A -85,B 0,C 180,E1 -28811.924,E2 -28811.924} C_VEL
LIN {X 0,Y 69.009,Z 263.062,A -85,B 0,C 180,E1 -28816.595,E2 -28816.595} C_VEL
LIN {X 0,Y 72.468,Z 269.041,A -85,B 0,C 180,E1 -28820.99,E2 -28820.99} C_VEL
LIN {X 0,Y 76.66,Z 277.554,A -85,B 0,C 180,E1 -28825.775,E2 -28825.775} C_VEL
LIN {X 0,Y 80.031,Z 288.891,A -85,B 0,C 180,E1 -28829.756,E2 -28829.756} C_VEL
LIN {X 0,Y 82.557,Z 298.941,A -85,B 0,C 180,E1 -28832.63,E2 -28832.63} C_VEL
LIN {X 0,Y 82.626,Z 318.978,A -85,B 0,C 180,E1 -28835.554,E2 -28835.554} C_VEL
LIN {X 0,Y 79.348,Z 346.877,A -85,B 0,C 180,E1 -28838.27,E2 -28838.27} C_VEL
LIN {X 0,Y 76.77,Z 361.059,A -85,B 0,C 180,E1 -28840.618,E2 -28840.618} C_VEL
LIN {X 0,Y 73.181,Z 374.389,A -85,B 0,C 180,E1 -28843.921,E2 -28843.921} C_VEL
LIN {X 0,Y 69.498,Z 385.731,A -85,B 0,C 180,E1 -28847.935,E2 -28847.935} C_VEL
LIN {X 0,Y 65.336,Z 397.25,A -85,B 0,C 180,E1 -28853.726,E2 -28853.726} C_VEL
LIN {X 0,Y 61.631,Z 407.57,A -85,B 0,C 180,E1 -28861.009,E2 -28861.009} C_VEL
LIN {X 0,Y 59.089,Z 416.026,A -85,B 0,C 180,E1 -28869.093,E2 -28869.093} C_VEL
LIN {X 0,Y 57.712,Z 423.031,A -85,B 0,C 180,E1 -28877.759,E2 -28877.759} C_VEL
LIN {X 0,Y 57.576,Z 428.728,A -85,B 0,C 180,E1 -28886.499,E2 -28886.499} C_VEL
LIN {X 0,Y 57.989,Z 432.484,A -85,B 0,C 180,E1 -28893.472,E2 -28893.472} C_VEL
LIN {X 0,Y 57.797,Z 436.55,A -85,B 0,C 180,E1 -28904.073,E2 -28904.073} C_VEL
LIN {X 0,Y 60.52,Z 440.496,A -85,B 0,C 180,E1 -28917.676,E2 -28917.676} C_VEL
LIN {X 0,Y 66.493,Z 443.073,A -85,B 0,C 180,E1 -28929.356,E2 -28929.356} C_VEL
LIN {X 0,Y 74.956,Z 444.343,A -85,B 0,C 180,E1 -28938.597,E2 -28938.597} C_VEL
LIN {X 0,Y 85.133,Z 444.335,A -85,B 0,C 180,E1 -28945.64,E2 -28945.64} C_VEL
LIN {X 0,Y 96.54,Z 443.04,A -85,B 0,C 180,E1 -28950.876,E2 -28950.876} C_VEL
LIN {X 0,Y 108.753,Z 440.435,A -85,B 0,C 180,E1 -28954.785,E2 -28954.785} C_VEL
LIN {X 0,Y 115.078,Z 438.61,A -85,B 0,C 180,E1 -28956.357,E2 -28956.357} C_VEL
LIN {X 0,Y 114.85,Z 438.636,A -85,B 0,C 180,E1 -28956.618,E2 -28956.618} C_VEL
LIN {X 0,Y 103.389,Z 440.803,A -85,B 0,C 180,E1 -28960.13,E2 -28960.13} C_VEL
LIN {X 0,Y 95.43,Z 441.59,A -85,B 0,C 180,E1 -28963.21,E2 -28963.21} C_VEL
LIN {X 0,Y 86.324,Z 441.658,A -85,B 0,C 180,E1 -28967.674,E2 -28967.674} C_VEL
LIN {X 0,Y 76.05,Z 440.407,A -85,B 0,C 180,E1 -28974.697,E2 -28974.697} C_VEL
LIN {X 0,Y 68.627,Z 438.259,A -85,B 0,C 180,E1 -28982.054,E2 -28982.054} C_VEL
LIN {X 0,Y 64.983,Z 436.867,A -85,B 0,C 180,E1 -28985.861,E2 -28985.861} C_VEL
LIN {X 0,Y 58.203,Z 433.926,A -85,B 0,C 180,E1 -28992.048,E2 -28992.048} C_VEL
LIN {X 0,Y 52.302,Z 430.259,A -85,B 0,C 180,E1 -28999.45,E2 -28999.45} C_VEL
LIN {X 0,Y 50.259,Z 427.678,A -85,B 0,C 180,E1 -29004.965,E2 -29004.965} C_VEL
LIN {X 0,Y 48.983,Z 421.764,A -85,B 0,C 180,E1 -29017.342,E2 -29017.342} C_VEL
LIN {X 0,Y 50.013,Z 413.922,A -85,B 0,C 180,E1 -29030.613,E2 -29030.613} C_VEL
LIN {X 0,Y 52.286,Z 405.831,A -85,B 0,C 180,E1 -29041.088,E2 -29041.088} C_VEL
LIN {X 0,Y 55.614,Z 396.801,A -85,B 0,C 180,E1 -29049.851,E2 -29049.851} C_VEL
LIN {X 0,Y 59.722,Z 386.419,A -85,B 0,C 180,E1 -29057.173,E2 -29057.173} C_VEL
LIN {X 0,Y 63.778,Z 375.492,A -85,B 0,C 180,E1 -29062.635,E2 -29062.635} C_VEL
LIN {X 0,Y 67.679,Z 363.501,A -85,B 0,C 180,E1 -29066.911,E2 -29066.911} C_VEL
LIN {X 0,Y 71.011,Z 351.135,A -85,B 0,C 180,E1 -29070.002,E2 -29070.002} C_VEL
LIN {X 0,Y 73.791,Z 336.912,A -85,B 0,C 180,E1 -29072.358,E2 -29072.358} C_VEL
LIN {X 0,Y 78.533,Z 298.674,A -85,B 0,C 180,E1 -29076.04,E2 -29076.04} C_VEL
LIN {X 0,Y 74.117,Z 285.587,A -85,B 0,C 180,E1 -29081.129,E2 -29081.129} C_VEL
LIN {X 0,Y 70.646,Z 276.881,A -85,B 0,C 180,E1 -29085.438,E2 -29085.438} C_VEL
LIN {X 0,Y 66.376,Z 269.314,A -85,B 0,C 180,E1 -29091.23,E2 -29091.23} C_VEL
LIN {X 0,Y 64.306,Z 266.325,A -85,B 0,C 180,E1 -29094.446,E2 -29094.446} C_VEL
LIN {X 0,Y 62.387,Z 263.355,A -85,B 0,C 180,E1 -29097.797,E2 -29097.797} C_VEL
LIN {X 0,Y 60.161,Z 260.308,A -85,B 0,C 180,E1 -29102.261,E2 -29102.261} C_VEL
LIN {X 0,Y 59.59,Z 259.149,A -85,B 0,C 180,E1 -29103.707,E2 -29103.707} C_VEL
LIN {X 0,Y 57.25,Z 256.905,A -85,B 0,C 180,E1 -29109.803,E2 -29109.803} C_VEL
LIN {X 0,Y 56.049,Z 254.074,A -85,B 0,C 180,E1 -29114.708,E2 -29114.708} C_VEL
LIN {X 0,Y 53.776,Z 252.837,A -85,B 0,C 180,E1 -29128.483,E2 -29128.483} C_VEL
LIN {X 0,Y 54.616,Z 253.074,A -85,B 0,C 180,E1 -29145.087,E2 -29145.087} C_VEL
LIN {X 0,Y 57.019,Z 254.079,A -85,B 0,C 180,E1 -29154.761,E2 -29154.761} C_VEL
LIN {X 0,Y 59.24,Z 258.14,A -85,B 0,C 180,E1 -29161.7,E2 -29161.7} C_VEL
LIN {X 0,Y 60.238,Z 259.352,A -85,B 0,C 180,E1 -29163.973,E2 -29163.973} C_VEL
LIN {X 0,Y 62.855,Z 263.91,A -85,B 0,C 180,E1 -29169.482,E2 -29169.482} C_VEL
LIN {X 0,Y 66.541,Z 270.258,A -85,B 0,C 180,E1 -29175.67,E2 -29175.67} C_VEL
LIN {X 0,Y 70.857,Z 278.936,A -85,B 0,C 180,E1 -29181.567,E2 -29181.567} C_VEL
LIN {X 0,Y 72.588,Z 283.444,A -85,B 0,C 180,E1 -29183.844,E2 -29183.844} C_VEL
LIN {X 0,Y 76.099,Z 297.213,A -85,B 0,C 180,E1 -29188.739,E2 -29188.739} C_VEL
LIN {X 0,Y 76.841,Z 301.378,A -85,B 0,C 180,E1 -29189.88,E2 -29189.88} C_VEL
LIN {X 0,Y 76.826,Z 318.607,A -85,B 0,C 180,E1 -29192.628,E2 -29192.628} C_VEL
LIN {X 0,Y 73.312,Z 346.679,A -85,B 0,C 180,E1 -29195.48,E2 -29195.48} C_VEL
LIN {X 0,Y 70.662,Z 360.438,A -85,B 0,C 180,E1 -29197.863,E2 -29197.863} C_VEL
LIN {X 0,Y 67.353,Z 372.252,A -85,B 0,C 180,E1 -29200.84,E2 -29200.84} C_VEL
LIN {X 0,Y 62.87,Z 385.376,A -85,B 0,C 180,E1 -29205.678,E2 -29205.678} C_VEL
LIN {X 0,Y 58.479,Z 396.856,A -85,B 0,C 180,E1 -29211.979,E2 -29211.979} C_VEL
LIN {X 0,Y 54.917,Z 406.198,A -85,B 0,C 180,E1 -29219.207,E2 -29219.207} C_VEL
LIN {X 0,Y 52.106,Z 414.941,A -85,B 0,C 180,E1 -29228.433,E2 -29228.433} C_VEL
LIN {X 0,Y 50.701,Z 421.945,A -85,B 0,C 180,E1 -29238.15,E2 -29238.15} C_VEL
LIN {X 0,Y 50.79,Z 428.675,A -85,B 0,C 180,E1 -29249.998,E2 -29249.998} C_VEL
LIN {X 0,Y 51.103,Z 430.551,A -85,B 0,C 180,E1 -29253.941,E2 -29253.941} C_VEL
LIN {X 0,Y 51.126,Z 434.831,A -85,B 0,C 180,E1 -29265.955,E2 -29265.955} C_VEL
LIN {X 0,Y 54.414,Z 439.122,A -85,B 0,C 180,E1 -29281.104,E2 -29281.104} C_VEL
LIN {X 0,Y 61.207,Z 441.943,A -85,B 0,C 180,E1 -29293.544,E2 -29293.544} C_VEL
LIN {X 0,Y 70.456,Z 443.478,A -85,B 0,C 180,E1 -29302.937,E2 -29302.937} C_VEL
LIN {X 0,Y 81.345,Z 443.768,A -85,B 0,C 180,E1 -29309.763,E2 -29309.763} C_VEL
LIN {X 0,Y 93.294,Z 442.813,A -85,B 0,C 180,E1 -29314.684,E2 -29314.684} C_VEL
LIN {X 0,Y 99.54,Z 441.856,A -85,B 0,C 180,E1 -29316.612,E2 -29316.612} C_VEL
LIN {X 0,Y 99.344,Z 441.845,A -85,B 0,C 180,E1 -29316.876,E2 -29316.876} C_VEL
LIN {X 0,Y 87.518,Z 442.353,A -85,B 0,C 180,E1 -29321.263,E2 -29321.263} C_VEL
LIN {X 0,Y 80.074,Z 441.98,A -85,B 0,C 180,E1 -29324.891,E2 -29324.891} C_VEL
LIN {X 0,Y 71.224,Z 440.62,A -85,B 0,C 180,E1 -29330.651,E2 -29330.651} C_VEL
LIN {X 0,Y 61.575,Z 437.566,A -85,B 0,C 180,E1 -29340,E2 -29340} C_VEL
LIN {X 0,Y 54.743,Z 433.41,A -85,B 0,C 180,E1 -29351.099,E2 -29351.099} C_VEL
LIN {X 0,Y 50.259,Z 427.678,A -85,B 0,C 180,E1 -29364.965,E2 -29364.965} C_VEL
LIN {X 0,Y 48.73,Z 424.931,A -85,B 0,C 180,E1 -29370.686,E2 -29370.686} C_VEL
LIN {X 0,Y 45.535,Z 419.714,A -85,B 0,C 180,E1 -29380.167,E2 -29380.167} C_VEL
LIN {X 0,Y 43.695,Z 415.044,A -85,B 0,C 180,E1 -29388.214,E2 -29388.214} C_VEL
LIN {X 0,Y 43.563,Z 411.27,A -85,B 0,C 180,E1 -29394.331,E2 -29394.331} C_VEL
LIN {X 0,Y 43.858,Z 409.964,A -85,B 0,C 180,E1 -29396.297,E2 -29396.297} C_VEL
LIN {X 0,Y 47.004,Z 401.021,A -85,B 0,C 180,E1 -29407.658,E2 -29407.658} C_VEL
LIN {X 0,Y 51.384,Z 390.486,A -85,B 0,C 180,E1 -29417.037,E2 -29417.037} C_VEL
LIN {X 0,Y 55.973,Z 379.286,A -85,B 0,C 180,E1 -29423.878,E2 -29423.878} C_VEL
LIN {X 0,Y 60.211,Z 367.823,A -85,B 0,C 180,E1 -29428.748,E2 -29428.748} C_VEL
LIN {X 0,Y 63.968,Z 355.504,A -85,B 0,C 180,E1 -29432.363,E2 -29432.363} C_VEL
LIN {X 0,Y 67.271,Z 341.642,A -85,B 0,C 180,E1 -29435.059,E2 -29435.059} C_VEL
LIN {X 0,Y 69.575,Z 326.169,A -85,B 0,C 180,E1 -29436.94,E2 -29436.94} C_VEL
LIN {X 0,Y 72.811,Z 300.235,A -85,B 0,C 180,E1 -29439.428,E2 -29439.428} C_VEL
LIN {X 0,Y 69.256,Z 289.133,A -85,B 0,C 180,E1 -29444.151,E2 -29444.151} C_VEL
LIN {X 0,Y 66.431,Z 281.469,A -85,B 0,C 180,E1 -29448.348,E2 -29448.348} C_VEL
LIN {X 0,Y 62.866,Z 274.562,A -85,B 0,C 180,E1 -29454.105,E2 -29454.105} C_VEL
LIN {X 0,Y 59.359,Z 269.136,A -85,B 0,C 180,E1 -29460.689,E2 -29460.689} C_VEL
LIN {X 0,Y 56.988,Z 265.4,A -85,B 0,C 180,E1 -29466.646,E2 -29466.646} C_VEL
LIN {X 0,Y 54.86,Z 262.595,A -85,B 0,C 180,E1 -29473.659,E2 -29473.659} C_VEL
LIN {X 0,Y 54.275,Z 260.904,A -85,B 0,C 180,E1 -29476.717,E2 -29476.717} C_VEL
LIN {X 0,Y 52.63,Z 259.908,A -85,B 0,C 180,E1 -29487.714,E2 -29487.714} C_VEL
LIN {X 0,Y 53.346,Z 260.037,A -85,B 0,C 180,E1 -29504.723,E2 -29504.723} C_VEL
LIN {X 0,Y 55.21,Z 260.882,A -85,B 0,C 180,E1 -29512.963,E2 -29512.963} C_VEL
LIN {X 0,Y 56.858,Z 264.314,A -85,B 0,C 180,E1 -29519.114,E2 -29519.114} C_VEL
LIN {X 0,Y 57.8,Z 265.765,A -85,B 0,C 180,E1 -29521.715,E2 -29521.715} C_VEL
LIN {X 0,Y 59.878,Z 269.697,A -85,B 0,C 180,E1 -29526.741,E2 -29526.741} C_VEL
LIN {X 0,Y 63.006,Z 275.596,A -85,B 0,C 180,E1 -29532.891,E2 -29532.891} C_VEL
LIN {X 0,Y 66.662,Z 283.662,A -85,B 0,C 180,E1 -29538.827,E2 -29538.827} C_VEL
LIN {X 0,Y 67.87,Z 287.046,A -85,B 0,C 180,E1 -29540.666,E2 -29540.666} C_VEL
LIN {X 0,Y 70.934,Z 300.299,A -85,B 0,C 180,E1 -29545.76,E2 -29545.76} C_VEL
LIN {X 0,Y 71.364,Z 303.317,A -85,B 0,C 180,E1 -29546.636,E2 -29546.636} C_VEL
LIN {X 0,Y 71.058,Z 319.728,A -85,B 0,C 180,E1 -29549.392,E2 -29549.392} C_VEL
LIN {X 0,Y 67.468,Z 346.496,A -85,B 0,C 180,E1 -29552.195,E2 -29552.195} C_VEL
LIN {X 0,Y 64.645,Z 360.25,A -85,B 0,C 180,E1 -29554.695,E2 -29554.695} C_VEL
LIN {X 0,Y 60.509,Z 373.789,A -85,B 0,C 180,E1 -29558.369,E2 -29558.369} C_VEL
LIN {X 0,Y 56.376,Z 385.032,A -85,B 0,C 180,E1 -29562.909,E2 -29562.909} C_VEL
LIN {X 0,Y 51.692,Z 396.43,A -85,B 0,C 180,E1 -29569.771,E2 -29569.771} C_VEL
LIN {X 0,Y 47.566,Z 406.649,A -85,B 0,C 180,E1 -29578.857,E2 -29578.857} C_VEL
LIN {X 0,Y 44.564,Z 416.171,A -85,B 0,C 180,E1 -29591.13,E2 -29591.13} C_VEL
LIN {X 0,Y 43.633,Z 424.259,A -85,B 0,C 180,E1 -29605.378,E2 -29605.378} C_VEL
LIN {X 0,Y 44.226,Z 428.507,A -85,B 0,C 180,E1 -29614.555,E2 -29614.555} C_VEL
LIN {X 0,Y 44.284,Z 432.084,A -85,B 0,C 180,E1 -29625.125,E2 -29625.125} C_VEL
LIN {X 0,Y 47.169,Z 436.6,A -85,B 0,C 180,E1 -29641.429,E2 -29641.429} C_VEL
LIN {X 0,Y 52.066,Z 439.312,A -85,B 0,C 180,E1 -29652.445,E2 -29652.445} C_VEL
LIN {X 0,Y 61.198,Z 441.813,A -85,B 0,C 180,E1 -29663.5,E2 -29663.5} C_VEL
LIN {X 0,Y 72.099,Z 443.019,A -85,B 0,C 180,E1 -29671.315,E2 -29671.315} C_VEL
LIN {X 0,Y 84.169,Z 442.997,A -85,B 0,C 180,E1 -29676.703,E2 -29676.703} C_VEL
LIN {X 0,Y 83.848,Z 442.942,A -85,B 0,C 180,E1 -29677.217,E2 -29677.217} C_VEL
LIN {X 0,Y 71.777,Z 441.707,A -85,B 0,C 180,E1 -29682.917,E2 -29682.917} C_VEL
LIN {X 0,Y 61.516,Z 439.298,A -85,B 0,C 180,E1 -29690.129,E2 -29690.129} C_VEL
LIN {X 0,Y 52.757,Z 435.648,A -85,B 0,C 180,E1 -29699.999,E2 -29699.999} C_VEL
LIN {X 0,Y 46.08,Z 430.583,A -85,B 0,C 180,E1 -29713.224,E2 -29713.224} C_VEL
LIN {X 0,Y 42.379,Z 423.815,A -85,B 0,C 180,E1 -29729.835,E2 -29729.835} C_VEL
LIN {X 0,Y 42.272,Z 416.515,A -85,B 0,C 180,E1 -29745.348,E2 -29745.348} C_VEL
LIN {X 0,Y 43.858,Z 409.964,A -85,B 0,C 180,E1 -29756.297,E2 -29756.297} C_VEL
LIN {X 0,Y 44.524,Z 406.009,A -85,B 0,C 180,E1 -29761.892,E2 -29761.892} C_VEL
LIN {X 0,Y 44.514,Z 398.949,A -85,B 0,C 180,E1 -29770.873,E2 -29770.873} C_VEL
LIN {X 0,Y 45.082,Z 391.373,A -85,B 0,C 180,E1 -29779.172,E2 -29779.172} C_VEL
LIN {X 0,Y 46.534,Z 386.553,A -85,B 0,C 180,E1 -29783.158,E2 -29783.158} C_VEL
LIN {X 0,Y 51.72,Z 374.322,A -85,B 0,C 180,E1 -29790.002,E2 -29790.002} C_VEL
LIN {X 0,Y 56.018,Z 362.548,A -85,B 0,C 180,E1 -29794.393,E2 -29794.393} C_VEL
LIN {X 0,Y 59.818,Z 349.59,A -85,B 0,C 180,E1 -29797.582,E2 -29797.582} C_VEL
LIN {X 0,Y 62.532,Z 336.967,A -85,B 0,C 180,E1 -29799.647,E2 -29799.647} C_VEL
LIN {X 0,Y 67.346,Z 302.076,A -85,B 0,C 180,E1 -29803.129,E2 -29803.129} C_VEL
LIN {X 0,Y 64.556,Z 292.515,A -85,B 0,C 180,E1 -29807.715,E2 -29807.715} C_VEL
LIN {X 0,Y 62.394,Z 286.011,A -85,B 0,C 180,E1 -29811.672,E2 -29811.672} C_VEL
LIN {X 0,Y 59.397,Z 279.746,A -85,B 0,C 180,E1 -29817.302,E2 -29817.302} C_VEL
LIN {X 0,Y 56.692,Z 275.139,A -85,B 0,C 180,E1 -29823.413,E2 -29823.413} C_VEL
LIN {X 0,Y 54.837,Z 271.817,A -85,B 0,C 180,E1 -29829.003,E2 -29829.003} C_VEL
LIN {X 0,Y 52.86,Z 268.719,A -85,B 0,C 180,E1 -29836.835,E2 -29836.835} C_VEL
LIN {X 0,Y 52.53,Z 267.708,A -85,B 0,C 180,E1 -29838.999,E2 -29838.999} C_VEL
LIN {X 0,Y 51.483,Z 266.972,A -85,B 0,C 180,E1 -29846.904,E2 -29846.904} C_VEL
LIN {X 0,Y 51.731,Z 266.933,A -85,B 0,C 180,E1 -29861.998,E2 -29861.998} C_VEL
LIN {X 0,Y 53.484,Z 267.88,A -85,B 0,C 180,E1 -29871.27,E2 -29871.27} C_VEL
LIN {X 0,Y 55.368,Z 271.946,A -85,B 0,C 180,E1 -29878.944,E2 -29878.944} C_VEL
LIN {X 0,Y 57.026,Z 275.55,A -85,B 0,C 180,E1 -29883.837,E2 -29883.837} C_VEL
LIN {X 0,Y 59.787,Z 281.267,A -85,B 0,C 180,E1 -29890.114,E2 -29890.114} C_VEL
LIN {X 0,Y 62.93,Z 289.127,A -85,B 0,C 180,E1 -29896.245,E2 -29896.245} C_VEL
LIN {X 0,Y 65.006,Z 298.478,A -85,B 0,C 180,E1 -29900.519,E2 -29900.519} C_VEL
LIN {X 0,Y 66.106,Z 304.45,A -85,B 0,C 180,E1 -29902.761,E2 -29902.761} C_VEL
LIN {X 0,Y 65.648,Z 319.938,A -85,B 0,C 180,E1 -29905.546,E2 -29905.546} C_VEL
LIN {X 0,Y 61.885,Z 346.155,A -85,B 0,C 180,E1 -29908.338,E2 -29908.338} C_VEL
LIN {X 0,Y 58.857,Z 359.797,A -85,B 0,C 180,E1 -29910.877,E2 -29910.877} C_VEL
LIN {X 0,Y 54.474,Z 373.247,A -85,B 0,C 180,E1 -29914.663,E2 -29914.663} C_VEL
LIN {X 0,Y 50.071,Z 384.438,A -85,B 0,C 180,E1 -29919.465,E2 -29919.465} C_VEL
LIN {X 0,Y 45.021,Z 395.801,A -85,B 0,C 180,E1 -29926.921,E2 -29926.921} C_VEL
LIN {X 0,Y 40.967,Z 405.088,A -85,B 0,C 180,E1 -29936.111,E2 -29936.111} C_VEL
LIN {X 0,Y 37.912,Z 413.594,A -85,B 0,C 180,E1 -29948.235,E2 -29948.235} C_VEL
LIN {X 0,Y 36.665,Z 420.59,A -85,B 0,C 180,E1 -29961.731,E2 -29961.731} C_VEL
LIN {X 0,Y 37.358,Z 426.356,A -85,B 0,C 180,E1 -29975.394,E2 -29975.394} C_VEL
LIN {X 0,Y 37.541,Z 429.326,A -85,B 0,C 180,E1 -29984.899,E2 -29984.899} C_VEL
LIN {X 0,Y 39.976,Z 433.748,A -85,B 0,C 180,E1 -30001.828,E2 -30001.828} C_VEL
LIN {X 0,Y 47.146,Z 437.902,A -85,B 0,C 180,E1 -30018.185,E2 -30018.185} C_VEL
LIN {X 0,Y 57.283,Z 440.648,A -85,B 0,C 180,E1 -30029.182,E2 -30029.182} C_VEL
LIN {X 0,Y 68.988,Z 442.143,A -85,B 0,C 180,E1 -30036.468,E2 -30036.468} C_VEL
LIN {X 0,Y 68.283,Z 441.917,A -85,B 0,C 180,E1 -30037.864,E2 -30037.864} C_VEL
LIN {X 0,Y 56.161,Z 438.861,A -85,B 0,C 180,E1 -30045.505,E2 -30045.505} C_VEL
LIN {X 0,Y 46.699,Z 434.776,A -85,B 0,C 180,E1 -30055.684,E2 -30055.684} C_VEL
LIN {X 0,Y 39.314,Z 429.275,A -85,B 0,C 180,E1 -30070.297,E2 -30070.297} C_VEL
LIN {X 0,Y 35.333,Z 422.102,A -85,B 0,C 180,E1 -30089.594,E2 -30089.594} C_VEL
LIN {X 0,Y 35.46,Z 414.319,A -85,B 0,C 180,E1 -30108.007,E2 -30108.007} C_VEL
LIN {X 0,Y 37.899,Z 406.277,A -85,B 0,C 180,E1 -30122.486,E2 -30122.486} C_VEL
LIN {X 0,Y 41.746,Z 397.058,A -85,B 0,C 180,E1 -30134.243,E2 -30134.243} C_VEL
LIN {X 0,Y 46.534,Z 386.553,A -85,B 0,C 180,E1 -30143.158,E2 -30143.158} C_VEL
LIN {X 0,Y 47.993,Z 381.733,A -85,B 0,C 180,E1 -30146.648,E2 -30146.648} C_VEL
LIN {X 0,Y 49.065,Z 373.44,A -85,B 0,C 180,E1 -30152.707,E2 -30152.707} C_VEL
LIN {X 0,Y 50.203,Z 364.597,A -85,B 0,C 180,E1 -30158.06,E2 -30158.06} C_VEL
LIN {X 0,Y 51.652,Z 358.995,A -85,B 0,C 180,E1 -30160.196,E2 -30160.196} C_VEL
LIN {X 0,Y 55.402,Z 346.011,A -85,B 0,C 180,E1 -30162.945,E2 -30162.945} C_VEL
LIN {X 0,Y 57.907,Z 333.537,A -85,B 0,C 180,E1 -30164.669,E2 -30164.669} C_VEL
LIN {X 0,Y 62.14,Z 303.703,A -85,B 0,C 180,E1 -30167.577,E2 -30167.577} C_VEL
LIN {X 0,Y 59.994,Z 295.318,A -85,B 0,C 180,E1 -30172.148,E2 -30172.148} C_VEL
LIN {X 0,Y 58.47,Z 290.423,A -85,B 0,C 180,E1 -30175.465,E2 -30175.465} C_VEL
LIN {X 0,Y 56.051,Z 284.759,A -85,B 0,C 180,E1 -30181.093,E2 -30181.093} C_VEL
LIN {X 0,Y 53.9,Z 280.688,A -85,B 0,C 180,E1 -30187.219,E2 -30187.219} C_VEL
LIN {X 0,Y 52.474,Z 277.877,A -85,B 0,C 180,E1 -30192.513,E2 -30192.513} C_VEL
LIN {X 0,Y 50.898,Z 274.484,A -85,B 0,C 180,E1 -30201.322,E2 -30201.322} C_VEL
LIN {X 0,Y 50.277,Z 273.953,A -85,B 0,C 180,E1 -30207.009,E2 -30207.009} C_VEL
LIN {X 0,Y 50.787,Z 273.999,A -85,B 0,C 180,E1 -30223.933,E2 -30223.933} C_VEL
LIN {X 0,Y 51.704,Z 274.581,A -85,B 0,C 180,E1 -30229.004,E2 -30229.004} C_VEL
LIN {X 0,Y 53.122,Z 278.17,A -85,B 0,C 180,E1 -30236.078,E2 -30236.078} C_VEL
LIN {X 0,Y 55.518,Z 284.119,A -85,B 0,C 180,E1 -30244.134,E2 -30244.134} C_VEL
LIN {X 0,Y 58.142,Z 290.956,A -85,B 0,C 180,E1 -30250.624,E2 -30250.624} C_VEL
LIN {X 0,Y 59.149,Z 294.517,A -85,B 0,C 180,E1 -30253.075,E2 -30253.075} C_VEL
LIN {X 0,Y 61.078,Z 305.913,A -85,B 0,C 180,E1 -30258.337,E2 -30258.337} C_VEL
LIN {X 0,Y 60.423,Z 320.574,A -85,B 0,C 180,E1 -30261.166,E2 -30261.166} C_VEL
LIN {X 0,Y 56.632,Z 345.363,A -85,B 0,C 180,E1 -30263.755,E2 -30263.755} C_VEL
LIN {X 0,Y 53.411,Z 359.121,A -85,B 0,C 180,E1 -30266.306,E2 -30266.306} C_VEL
LIN {X 0,Y 48.741,Z 372.599,A -85,B 0,C 180,E1 -30270.096,E2 -30270.096} C_VEL
LIN {X 0,Y 43.992,Z 383.789,A -85,B 0,C 180,E1 -30275.036,E2 -30275.036} C_VEL
LIN {X 0,Y 38.52,Z 395.187,A -85,B 0,C 180,E1 -30283.126,E2 -30283.126} C_VEL
LIN {X 0,Y 33.646,Z 405.412,A -85,B 0,C 180,E1 -30294.94,E2 -30294.94} C_VEL
LIN {X 0,Y 30.41,Z 414.693,A -85,B 0,C 180,E1 -30311.983,E2 -30311.983} C_VEL
LIN {X 0,Y 30.243,Z 422.928,A -85,B 0,C 180,E1 -30333.327,E2 -30333.327} C_VEL
LIN {X 0,Y 30.874,Z 425.969,A -85,B 0,C 180,E1 -30343.154,E2 -30343.154} C_VEL
LIN {X 0,Y 34.326,Z 431.932,A -85,B 0,C 180,E1 -30367.892,E2 -30367.892} C_VEL
LIN {X 0,Y 42.824,Z 436.312,A -85,B 0,C 180,E1 -30385.138,E2 -30385.138} C_VEL
LIN {X 0,Y 54.016,Z 439.384,A -85,B 0,C 180,E1 -30395.606,E2 -30395.606} C_VEL
LIN {X 0,Y 55.024,Z 439.489,A -85,B 0,C 180,E1 -30397.469,E2 -30397.469} C_VEL
LIN {X 0,Y 43.208,Z 434.898,A -85,B 0,C 180,E1 -30407.394,E2 -30407.394} C_VEL
LIN {X 0,Y 35.138,Z 429.915,A -85,B 0,C 180,E1 -30420.068,E2 -30420.068} C_VEL
LIN {X 0,Y 29.63,Z 423.731,A -85,B 0,C 180,E1 -30438.433,E2 -30438.433} C_VEL
LIN {X 0,Y 28.044,Z 416.086,A -85,B 0,C 180,E1 -30461.258,E2 -30461.258} C_VEL
LIN {X 0,Y 29.801,Z 408.746,A -85,B 0,C 180,E1 -30479.003,E2 -30479.003} C_VEL
LIN {X 0,Y 34.08,Z 398.774,A -85,B 0,C 180,E1 -30495.457,E2 -30495.457} C_VEL
LIN {X 0,Y 39.539,Z 387.932,A -85,B 0,C 180,E1 -30506.493,E2 -30506.493} C_VEL
LIN {X 0,Y 45.091,Z 376.053,A -85,B 0,C 180,E1 -30513.912,E2 -30513.912} C_VEL
LIN {X 0,Y 49.747,Z 364.541,A -85,B 0,C 180,E1 -30518.542,E2 -30518.542} C_VEL
LIN {X 0,Y 51.652,Z 358.995,A -85,B 0,C 180,E1 -30520.196,E2 -30520.196} C_VEL
LIN {X 0,Y 52.897,Z 353.469,A -85,B 0,C 180,E1 -30522.071,E2 -30522.071} C_VEL
LIN {X 0,Y 53.242,Z 344.221,A -85,B 0,C 180,E1 -30525.994,E2 -30525.994} C_VEL
LIN {X 0,Y 53.282,Z 334.783,A -85,B 0,C 180,E1 -30529.487,E2 -30529.487} C_VEL
LIN {X 0,Y 53.826,Z 328.951,A -85,B 0,C 180,E1 -30530.532,E2 -30530.532} C_VEL
LIN {X 0,Y 57.345,Z 305.424,A -85,B 0,C 180,E1 -30532.694,E2 -30532.694} C_VEL
LIN {X 0,Y 55.487,Z 297.301,A -85,B 0,C 180,E1 -30537.787,E2 -30537.787} C_VEL
LIN {X 0,Y 54.508,Z 294.002,A -85,B 0,C 180,E1 -30540.579,E2 -30540.579} C_VEL
LIN {X 0,Y 53.026,Z 289.997,A -85,B 0,C 180,E1 -30545.142,E2 -30545.142} C_VEL
LIN {X 0,Y 51.239,Z 286.013,A -85,B 0,C 180,E1 -30551.745,E2 -30551.745} C_VEL
LIN {X 0,Y 50.494,Z 284.253,A -85,B 0,C 180,E1 -30555.28,E2 -30555.28} C_VEL
LIN {X 0,Y 49.45,Z 281.431,A -85,B 0,C 180,E1 -30562.832,E2 -30562.832} C_VEL
LIN {X 0,Y 48.93,Z 280.915,A -85,B 0,C 180,E1 -30569.525,E2 -30569.525} C_VEL
LIN {X 0,Y 49.851,Z 281.158,A -85,B 0,C 180,E1 -30585.764,E2 -30585.764} C_VEL
LIN {X 0,Y 50.8,Z 283.597,A -85,B 0,C 180,E1 -30591.676,E2 -30591.676} C_VEL
LIN {X 0,Y 52.67,Z 289.584,A -85,B 0,C 180,E1 -30600.38,E2 -30600.38} C_VEL
LIN {X 0,Y 54.708,Z 296.107,A -85,B 0,C 180,E1 -30606.945,E2 -30606.945} C_VEL
LIN {X 0,Y 55.472,Z 300.076,A -85,B 0,C 180,E1 -30609.485,E2 -30609.485} C_VEL
LIN {X 0,Y 56.472,Z 308.479,A -85,B 0,C 180,E1 -30613.472,E2 -30613.472} C_VEL
LIN {X 0,Y 55.607,Z 321.356,A -85,B 0,C 180,E1 -30616.031,E2 -30616.031} C_VEL
LIN {X 0,Y 51.816,Z 344.59,A -85,B 0,C 180,E1 -30618.291,E2 -30618.291} C_VEL
LIN {X 0,Y 48.377,Z 358.431,A -85,B 0,C 180,E1 -30620.732,E2 -30620.732} C_VEL
LIN {X 0,Y 44.148,Z 370.118,A -85,B 0,C 180,E1 -30623.739,E2 -30623.739} C_VEL
LIN {X 0,Y 38.994,Z 381.623,A -85,B 0,C 180,E1 -30628.516,E2 -30628.516} C_VEL
LIN {X 0,Y 32.874,Z 393.316,A -85,B 0,C 180,E1 -30636.702,E2 -30636.702} C_VEL
LIN {X 0,Y 27.277,Z 403.693,A -85,B 0,C 180,E1 -30649.904,E2 -30649.904} C_VEL
LIN {X 0,Y 23.612,Z 412.64,A -85,B 0,C 180,E1 -30669.516,E2 -30669.516} C_VEL
LIN {X 0,Y 23.318,Z 420.412,A -85,B 0,C 180,E1 -30694.317,E2 -30694.317} C_VEL
LIN {X 0,Y 24.354,Z 423.704,A -85,B 0,C 180,E1 -30706.768,E2 -30706.768} C_VEL
LIN {X 0,Y 27.221,Z 428.426,A -85,B 0,C 180,E1 -30729.234,E2 -30729.234} C_VEL
LIN {X 0,Y 36.48,Z 433.616,A -85,B 0,C 180,E1 -30750.098,E2 -30750.098} C_VEL
LIN {X 0,Y 39.282,Z 434.673,A -85,B 0,C 180,E1 -30753.444,E2 -30753.444} C_VEL
LIN {X 0,Y 41.228,Z 435.199,A -85,B 0,C 180,E1 -30757.452,E2 -30757.452} C_VEL
LIN {X 0,Y 32.433,Z 430.588,A -85,B 0,C 180,E1 -30767.484,E2 -30767.484} C_VEL
LIN {X 0,Y 24.027,Z 423.527,A -85,B 0,C 180,E1 -30788.409,E2 -30788.409} C_VEL
LIN {X 0,Y 21.052,Z 416.143,A -85,B 0,C 180,E1 -30815.741,E2 -30815.741} C_VEL
LIN {X 0,Y 22.649,Z 408.461,A -85,B 0,C 180,E1 -30840.457,E2 -30840.457} C_VEL
LIN {X 0,Y 27.436,Z 398.598,A -85,B 0,C 180,E1 -30860.349,E2 -30860.349} C_VEL
LIN {X 0,Y 33.267,Z 388.105,A -85,B 0,C 180,E1 -30872.169,E2 -30872.169} C_VEL
LIN {X 0,Y 39.781,Z 375.375,A -85,B 0,C 180,E1 -30880.179,E2 -30880.179} C_VEL
LIN {X 0,Y 44.856,Z 363.494,A -85,B 0,C 180,E1 -30884.669,E2 -30884.669} C_VEL
LIN {X 0,Y 49.603,Z 349.207,A -85,B 0,C 180,E1 -30887.952,E2 -30887.952} C_VEL
LIN {X 0,Y 52.713,Z 335.881,A -85,B 0,C 180,E1 -30889.814,E2 -30889.814} C_VEL
LIN {X 0,Y 53.826,Z 328.951,A -85,B 0,C 180,E1 -30890.532,E2 -30890.532} C_VEL
LIN {X 0,Y 54.031,Z 325.06,A -85,B 0,C 180,E1 -30891.384,E2 -30891.384} C_VEL
LIN {X 0,Y 53.21,Z 318.953,A -85,B 0,C 180,E1 -30894.347,E2 -30894.347} C_VEL
LIN {X 0,Y 52.512,Z 312.846,A -85,B 0,C 180,E1 -30897.435,E2 -30897.435} C_VEL
LIN {X 0,Y 52.779,Z 308.951,A -85,B 0,C 180,E1 -30898.333,E2 -30898.333} C_VEL
LIN {X 0,Y 52.975,Z 306.955,A -85,B 0,C 180,E1 -30898.697,E2 -30898.697} C_VEL
LIN {X 0,Y 51.624,Z 299.721,A -85,B 0,C 180,E1 -30904.123,E2 -30904.123} C_VEL
LIN {X 0,Y 50.342,Z 295.367,A -85,B 0,C 180,E1 -30909.381,E2 -30909.381} C_VEL
LIN {X 0,Y 48.75,Z 290.823,A -85,B 0,C 180,E1 -30917.61,E2 -30917.61} C_VEL
LIN {X 0,Y 47.988,Z 288.164,A -85,B 0,C 180,E1 -30925.216,E2 -30925.216} C_VEL
LIN {X 0,Y 47.622,Z 287.835,A -85,B 0,C 180,E1 -30933.722,E2 -30933.722} C_VEL
LIN {X 0,Y 48.384,Z 288.036,A -85,B 0,C 180,E1 -30944.22,E2 -30944.22} C_VEL
LIN {X 0,Y 48.971,Z 290.468,A -85,B 0,C 180,E1 -30949.401,E2 -30949.401} C_VEL
LIN {X 0,Y 50.425,Z 296.497,A -85,B 0,C 180,E1 -30957.998,E2 -30957.998} C_VEL
LIN {X 0,Y 51.541,Z 301.594,A -85,B 0,C 180,E1 -30962.991,E2 -30962.991} C_VEL
LIN {X 0,Y 52.291,Z 309.634,A -85,B 0,C 180,E1 -30967.496,E2 -30967.496} C_VEL
LIN {X 0,Y 51.387,Z 321.017,A -85,B 0,C 180,E1 -30969.929,E2 -30969.929} C_VEL
LIN {X 0,Y 47.367,Z 344.244,A -85,B 0,C 180,E1 -30971.934,E2 -30971.934} C_VEL
LIN {X 0,Y 43.91,Z 357.308,A -85,B 0,C 180,E1 -30973.982,E2 -30973.982} C_VEL
LIN {X 0,Y 39.423,Z 369.114,A -85,B 0,C 180,E1 -30976.614,E2 -30976.614} C_VEL
LIN {X 0,Y 33.863,Z 380.685,A -85,B 0,C 180,E1 -30980.934,E2 -30980.934} C_VEL
LIN {X 0,Y 27.1,Z 392.45,A -85,B 0,C 180,E1 -30988.915,E2 -30988.915} C_VEL
LIN {X 0,Y 21.259,Z 401.907,A -85,B 0,C 180,E1 -31001.828,E2 -31001.828} C_VEL
LIN {X 0,Y 16.89,Z 410.61,A -85,B 0,C 180,E1 -31025.404,E2 -31025.404} C_VEL
LIN {X 0,Y 16.894,Z 419.011,A -85,B 0,C 180,E1 -31061.999,E2 -31061.999} C_VEL
LIN {X 0,Y 18.051,Z 421.286,A -85,B 0,C 180,E1 -31072.907,E2 -31072.907} C_VEL
LIN {X 0,Y 25.013,Z 427.884,A -85,B 0,C 180,E1 -31107.444,E2 -31107.444} C_VEL
LIN {X 0,Y 26.609,Z 428.727,A -85,B 0,C 180,E1 -31110.692,E2 -31110.692} C_VEL
LIN {X 0,Y 28.812,Z 429.721,A -85,B 0,C 180,E1 -31116.183,E2 -31116.183} C_VEL
LIN {X 0,Y 19.758,Z 423.462,A -85,B 0,C 180,E1 -31132.574,E2 -31132.574} C_VEL
LIN {X 0,Y 14.244,Z 415.255,A -85,B 0,C 180,E1 -31169.561,E2 -31169.561} C_VEL
LIN {X 0,Y 16.146,Z 406.789,A -85,B 0,C 180,E1 -31207.655,E2 -31207.655} C_VEL
LIN {X 0,Y 21.796,Z 397.239,A -85,B 0,C 180,E1 -31230.005,E2 -31230.005} C_VEL
LIN {X 0,Y 28.724,Z 386.242,A -85,B 0,C 180,E1 -31241.855,E2 -31241.855} C_VEL
LIN {X 0,Y 35.35,Z 374.137,A -85,B 0,C 180,E1 -31248.464,E2 -31248.464} C_VEL
LIN {X 0,Y 40.564,Z 362.4,A -85,B 0,C 180,E1 -31252.147,E2 -31252.147} C_VEL
LIN {X 0,Y 45.226,Z 348.979,A -85,B 0,C 180,E1 -31254.675,E2 -31254.675} C_VEL
LIN {X 0,Y 48.325,Z 336.165,A -85,B 0,C 180,E1 -31256.161,E2 -31256.161} C_VEL
LIN {X 0,Y 52.779,Z 308.951,A -85,B 0,C 180,E1 -31258.333,E2 -31258.333} C_VEL
LIN {X 0,Y 52.782,Z 306.693,A -85,B 0,C 180,E1 -31259.137,E2 -31259.137} C_VEL
LIN {X 0,Y 52.08,Z 304.415,A -85,B 0,C 180,E1 -31261.308,E2 -31261.308} C_VEL
LIN {X 0,Y 50.548,Z 302.258,A -85,B 0,C 180,E1 -31265.494,E2 -31265.494} C_VEL
LIN {X 0,Y 47.451,Z 298.95,A -85,B 0,C 180,E1 -31276.962,E2 -31276.962} C_VEL
LIN {X 0,Y 47.219,Z 298.276,A -85,B 0,C 180,E1 -31278.608,E2 -31278.608} C_VEL
LIN {X 0,Y 46.625,Z 295.057,A -85,B 0,C 180,E1 -31287.184,E2 -31287.184} C_VEL
LIN {X 0,Y 46.431,Z 294.847,A -85,B 0,C 180,E1 -31295.261,E2 -31295.261} C_VEL
LIN {X 0,Y 46.96,Z 295.205,A -85,B 0,C 180,E1 -31303.014,E2 -31303.014} C_VEL
LIN {X 0,Y 47.692,Z 300.242,A -85,B 0,C 180,E1 -31311.294,E2 -31311.294} C_VEL
LIN {X 0,Y 48.464,Z 305.469,A -85,B 0,C 180,E1 -31317.16,E2 -31317.16} C_VEL
LIN {X 0,Y 48.625,Z 312.26,A -85,B 0,C 180,E1 -31321.028,E2 -31321.028} C_VEL
LIN {X 0,Y 47.522,Z 322.245,A -85,B 0,C 180,E1 -31322.989,E2 -31322.989} C_VEL
LIN {X 0,Y 43.477,Z 344.264,A -85,B 0,C 180,E1 -31324.433,E2 -31324.433} C_VEL
LIN {X 0,Y 39.754,Z 357.383,A -85,B 0,C 180,E1 -31326.027,E2 -31326.027} C_VEL
LIN {X 0,Y 34.61,Z 369.901,A -85,B 0,C 180,E1 -31328.111,E2 -31328.111} C_VEL
LIN {X 0,Y 27.848,Z 382.667,A -85,B 0,C 180,E1 -31332.037,E2 -31332.037} C_VEL
LIN {X 0,Y 20.337,Z 394.055,A -85,B 0,C 180,E1 -31339.63,E2 -31339.63} C_VEL
LIN {X 0,Y 12.946,Z 404.279,A -85,B 0,C 180,E1 -31358.431,E2 -31358.431} C_VEL
LIN {X 0,Y 9.303,Z 412.047,A -85,B 0,C 180,E1 -31399.102,E2 -31399.102} C_VEL
LIN {X 0,Y 12.145,Z 418.692,A -85,B 0,C 180,E1 -31445.347,E2 -31445.347} C_VEL
LIN {X 0,Y 16.338,Z 422.44,A -85,B 0,C 180,E1 -31469.337,E2 -31469.337} C_VEL
LIN {X 0,Y 15.883,Z 422.083,A -85,B 0,C 180,E1 -31473.735,E2 -31473.735} C_VEL
LIN {X 0,Y 7.78,Z 414.069,A -85,B 0,C 180,E1 -31514.919,E2 -31514.919} C_VEL
LIN {X 0,Y 9.457,Z 406.055,A -85,B 0,C 180,E1 -31578.735,E2 -31578.735} C_VEL
LIN {X 0,Y 16.483,Z 396.612,A -85,B 0,C 180,E1 -31604.154,E2 -31604.154} C_VEL
LIN {X 0,Y 23.958,Z 386.102,A -85,B 0,C 180,E1 -31613.551,E2 -31613.551} C_VEL
LIN {X 0,Y 30.687,Z 374.831,A -85,B 0,C 180,E1 -31618.222,E2 -31618.222} C_VEL
LIN {X 0,Y 36.684,Z 362.233,A -85,B 0,C 180,E1 -31620.993,E2 -31620.993} C_VEL
LIN {X 0,Y 41.612,Z 348.584,A -85,B 0,C 180,E1 -31622.732,E2 -31622.732} C_VEL
LIN {X 0,Y 44.808,Z 335.547,A -85,B 0,C 180,E1 -31623.74,E2 -31623.74} C_VEL
LIN {X 0,Y 49.281,Z 308.968,A -85,B 0,C 180,E1 -31625.47,E2 -31625.47} C_VEL
LIN {X 0,Y 48.583,Z 303.773,A -85,B 0,C 180,E1 -31629.923,E2 -31629.923} C_VEL
LIN {X 0,Y 47.869,Z 300.803,A -85,B 0,C 180,E1 -31633.963,E2 -31633.963} C_VEL
LIN {X 0,Y 47.219,Z 298.276,A -85,B 0,C 180,E1 -31638.608,E2 -31638.608} C_VEL
LIN {X 0,Y 46.775,Z 298.11,A -85,B 0,C 180,E1 -31641.305,E2 -31641.305} C_VEL
LIN {X 0,Y 46.105,Z 299.448,A -85,B 0,C 180,E1 -31644.736,E2 -31644.736} C_VEL
LIN {X 0,Y 45.339,Z 301.698,A -85,B 0,C 180,E1 -31649.894,E2 -31649.894} C_VEL
LIN {X 0,Y 45.247,Z 301.853,A -85,B 0,C 180,E1 -31651.52,E2 -31651.52} C_VEL
LIN {X 0,Y 45.476,Z 302.181,A -85,B 0,C 180,E1 -31660.617,E2 -31660.617} C_VEL
LIN {X 0,Y 45.733,Z 307.188,A -85,B 0,C 180,E1 -31668.222,E2 -31668.222} C_VEL
LIN {X 0,Y 45.857,Z 309.512,A -85,B 0,C 180,E1 -31670.64,E2 -31670.64} C_VEL
LIN {X 0,Y 45.729,Z 314.275,A -85,B 0,C 180,E1 -31673.446,E2 -31673.446} C_VEL
LIN {X 0,Y 44.628,Z 322.539,A -85,B 0,C 180,E1 -31674.931,E2 -31674.931} C_VEL
LIN {X 0,Y 40.531,Z 343.959,A -85,B 0,C 180,E1 -31675.629,E2 -31675.629} C_VEL
LIN {X 0,Y 36.531,Z 357.308,A -85,B 0,C 180,E1 -31676.431,E2 -31676.431} C_VEL
LIN {X 0,Y 30.786,Z 370.527,A -85,B 0,C 180,E1 -31677.2,E2 -31677.2} C_VEL
LIN {X 0,Y 24.609,Z 381.555,A -85,B 0,C 180,E1 -31678.429,E2 -31678.429} C_VEL
LIN {X 0,Y 16.395,Z 393.148,A -85,B 0,C 180,E1 -31681.264,E2 -31681.264} C_VEL
LIN {X 0,Y 7.207,Z 403.769,A -85,B 0,C 180,E1 -31692.738,E2 -31692.738} C_VEL
LIN {X 0,Y 2.463,Z 410.32,A -85,B 0,C 180,E1 -31769.955,E2 -31769.955} C_VEL
LIN {X 0,Y 1.848,Z 410.864,A -85,B 0,C 180,E1 -31818.211,E2 -31818.211} C_VEL
LIN {X 0,Y 7.595,Z 402.027,A -85,B 0,C 180,E1 -31985.953,E2 -31985.953} C_VEL
LIN {X 0,Y 16.305,Z 391.823,A -85,B 0,C 180,E1 -31989.264,E2 -31989.264} C_VEL
LIN {X 0,Y 24.374,Z 380.19,A -85,B 0,C 180,E1 -31990.506,E2 -31990.506} C_VEL
LIN {X 0,Y 31,Z 368.095,A -85,B 0,C 180,E1 -31991.235,E2 -31991.235} C_VEL
LIN {X 0,Y 36.578,Z 354.84,A -85,B 0,C 180,E1 -31991.874,E2 -31991.874} C_VEL
LIN {X 0,Y 40.586,Z 341.596,A -85,B 0,C 180,E1 -31992.126,E2 -31992.126} C_VEL
LIN {X 0,Y 44.91,Z 318.737,A -85,B 0,C 180,E1 -31992.834,E2 -31992.834} C_VEL
LIN {X 0,Y 46.224,Z 310.903,A -85,B 0,C 180,E1 -31993.268,E2 -31993.268} C_VEL
LIN {X 0,Y 45.964,Z 307.594,A -85,B 0,C 180,E1 -31996.707,E2 -31996.707} C_VEL
LIN {X 0,Y 45.419,Z 303.644,A -85,B 0,C 180,E1 -32004.153,E2 -32004.153} C_VEL
LIN {X 0,Y 45.317,Z 301.933,A -85,B 0,C 180,E1 -32009.4,E2 -32009.4} C_VEL
LIN {X 0,Y 45.247,Z 301.853,A -85,B 0,C 180,E1 -32011.52,E2 -32011.52} C_VEL
LIN {X 0,Y 45.095,Z 302.53,A -85,B 0,C 180,E1 -32013.761,E2 -32013.761} C_VEL
LIN {X 0,Y 44.665,Z 305.274,A -85,B 0,C 180,E1 -32016.301,E2 -32016.301} C_VEL
LIN {X 0,Y 44.002,Z 310.137,A -85,B 0,C 180,E1 -32019.529,E2 -32019.529} C_VEL
LIN {X 0,Y 43.96,Z 310.704,A -85,B 0,C 180,E1 -32020.222,E2 -32020.222} C_VEL
LIN {X 0,Y 43.829,Z 313.409,A -85,B 0,C 180,E1 -32023.389,E2 -32023.389} C_VEL
LIN {X 0,Y 43.572,Z 316.119,A -85,B 0,C 180,E1 -32024.957,E2 -32024.957} C_VEL
LIN {X 0,Y 42.489,Z 323.149,A -85,B 0,C 180,E1 -32025.977,E2 -32025.977} C_VEL
LIN {X 0,Y 38.494,Z 343.677,A -85,B 0,C 180,E1 -32025.768,E2 -32025.768} C_VEL
LIN {X 0,Y 34.49,Z 356.862,A -85,B 0,C 180,E1 -32025.46,E2 -32025.46} C_VEL
LIN {X 0,Y 29.217,Z 369.162,A -85,B 0,C 180,E1 -32024.207,E2 -32024.207} C_VEL
LIN {X 0,Y 22.805,Z 380.811,A -85,B 0,C 180,E1 -32021.822,E2 -32021.822} C_VEL
LIN {X 0,Y 15.351,Z 391.692,A -85,B 0,C 180,E1 -32016.313,E2 -32016.313} C_VEL
LIN {X 0,Y 16.112,Z 390.606,A -85,B 0,C 180,E1 -32014.141,E2 -32014.141} C_VEL
LIN {X 0,Y 23.677,Z 378.861,A -85,B 0,C 180,E1 -32007.092,E2 -32007.092} C_VEL
LIN {X 0,Y 30.048,Z 366.67,A -85,B 0,C 180,E1 -32004.225,E2 -32004.225} C_VEL
LIN {X 0,Y 35.296,Z 353.463,A -85,B 0,C 180,E1 -32002.799,E2 -32002.799} C_VEL
LIN {X 0,Y 39.242,Z 339.63,A -85,B 0,C 180,E1 -32001.925,E2 -32001.925} C_VEL
LIN {X 0,Y 44.043,Z 313.179,A -85,B 0,C 180,E1 -32001.842,E2 -32001.842} C_VEL
LIN {X 0,Y 44.003,Z 309.811,A -85,B 0,C 180,E1 -32008.383,E2 -32008.383} C_VEL
LIN {X 0,Y 44.045,Z 308.844,A -85,B 0,C 180,E1 -32011.4,E2 -32011.4} C_VEL
LIN {X 0,Y 44.052,Z 309.092,A -85,B 0,C 180,E1 -32017.438,E2 -32017.438} C_VEL
LIN {X 0,Y 43.96,Z 310.704,A -85,B 0,C 180,E1 -32020.222,E2 -32020.222} C_VEL
LIN {X 0,Y 43.745,Z 313.371,A -85,B 0,C 180,E1 -32022.534,E2 -32022.534} C_VEL
LIN {X 0,Y 43.212,Z 317.452,A -85,B 0,C 180,E1 -32023.659,E2 -32023.659} C_VEL
LIN {X 0,Y 42.158,Z 323.254,A -85,B 0,C 180,E1 -32022.878,E2 -32022.878} C_VEL
LIN {X 0,Y 39.044,Z 337.589,A -85,B 0,C 180,E1 -32016.26,E2 -32016.26} C_VEL
LIN {X 0,Y 38.065,Z 341.857,A -85,B 0,C 180,E1 -32015.223,E2 -32015.223} C_VEL
LIN {X 0,Y 36.012,Z 349.671,A -85,B 0,C 180,E1 -32014.509,E2 -32014.509} C_VEL
LIN {X 0,Y 35.991,Z 349.725,A -85,B 0,C 180,E1 -32013.793,E2 -32013.793} C_VEL
LIN {X 0,Y 39.172,Z 336.607,A -85,B 0,C 180,E1 -32012.206,E2 -32012.206} C_VEL
LIN {X 0,Y 42.715,Z 316.534,A -85,B 0,C 180,E1 -32011.355,E2 -32011.355} C_VEL
LIN {X 0,Y 42.794,Z 315.86,A -85,B 0,C 180,E1 -32013.333,E2 -32013.333} C_VEL
LIN {X 0,Y 42.71,Z 316.365,A -85,B 0,C 180,E1 -32014.682,E2 -32014.682} C_VEL
LIN {X 0,Y 42.567,Z 317.29,A -85,B 0,C 180,E1 -32015.637,E2 -32015.637} C_VEL
LIN {X 0,Y 41.706,Z 322.394,A -85,B 0,C 180,E1 -32016.408,E2 -32016.408} C_VEL
LIN {X 0,Y 38.065,Z 341.857,A -85,B 0,C 180,E1 -32015.223,E2 -32015.223} C_VEL
LIN {X 0,Y 38.008,Z 342.34,A -85,B 0,C 180,E1 -32015.199,E2 -32015.199} C_VEL
LIN {X 0,Y 38.008,Z 600,A -85,B 0,C 180,E1 -32015.199,E2 -32015.199} C_VEL
LIN {X 0,Y 38.008,Z 600,A -85,B 0,C 180,E1 -32015.199,E2 -32015.199}

QRS_NEXT_CUT()

QRS_NEXT()
QRS_HOME()

END
